LIN {X 0,Y 523.367,Z 631.707,A -85,B 0,C 180,E1 -4773.079,E2 -4773.079} C_VEL
LIN {X 0,Y 523.424,Z 628.783,A -85,B 0,C 180,E1 -4774.235,E2 -4774.235} C_VEL
LIN {X 0,Y 523.464,Z 624.823,A -85,B 0,C 180,E1 -4775.393,E2 -4775.393} C_VEL
LIN {X 0,Y 523.519,Z 619.605,A -85,B 0,C 180,E1 -4776.577,E2 -4776.577} C_VEL
LIN {X 0,Y 523.664,Z 613.306,A -85,B 0,C 180,E1 -4777.713,E2 -4777.713} C_VEL
LIN {X 0,Y 523.85,Z 605.295,A -85,B 0,C 180,E1 -4778.875,E2 -4778.875} C_VEL
LIN {X 0,Y 524.066,Z 597.13,A -85,B 0,C 180,E1 -4779.845,E2 -4779.845} C_VEL
LIN {X 0,Y 524.349,Z 587.171,A -85,B 0,C 180,E1 -4780.815,E2 -4780.815} C_VEL
LIN {X 0,Y 524.625,Z 575.842,A -85,B 0,C 180,E1 -4781.695,E2 -4781.695} C_VEL
LIN {X 0,Y 524.913,Z 564.896,A -85,B 0,C 180,E1 -4782.37,E2 -4782.37} C_VEL
LIN {X 0,Y 525.171,Z 552.673,A -85,B 0,C 180,E1 -4782.953,E2 -4782.953} C_VEL
LIN {X 0,Y 525.375,Z 539.835,A -85,B 0,C 180,E1 -4783.391,E2 -4783.391} C_VEL
LIN {X 0,Y 525.592,Z 526.212,A -85,B 0,C 180,E1 -4783.681,E2 -4783.681} C_VEL
LIN {X 0,Y 525.826,Z 432.447,A -85,B 0,C 180,E1 -4784.974,E2 -4784.974} C_VEL
LIN {X 0,Y 524.297,Z 423.023,A -85,B 0,C 180,E1 -4785.174,E2 -4785.174} C_VEL
LIN {X 0,Y 524.677,Z 405.609,A -85,B 0,C 180,E1 -4788.003,E2 -4788.003} C_VEL
LIN {X 0,Y 525.177,Z 385.391,A -85,B 0,C 180,E1 -4791.387,E2 -4791.387} C_VEL
LIN {X 0,Y 525.133,Z 380.293,A -85,B 0,C 180,E1 -4792.258,E2 -4792.258} C_VEL
LIN {X 0,Y 523.971,Z 373.816,A -85,B 0,C 180,E1 -4793.465,E2 -4793.465} C_VEL
LIN {X 0,Y 523.976,Z 373.714,A -85,B 0,C 180,E1 -4796.271,E2 -4796.271} C_VEL
LIN {X 0,Y 523.956,Z 373.722,A -85,B 0,C 180,E1 -4799.323,E2 -4799.323} C_VEL
LIN {X 0,Y 523.941,Z 373.716,A -85,B 0,C 180,E1 -4802.449,E2 -4802.449} C_VEL
LIN {X 0,Y 523.936,Z 373.723,A -85,B 0,C 180,E1 -4805.225,E2 -4805.225} C_VEL
LIN {X 0,Y 523.919,Z 373.719,A -85,B 0,C 180,E1 -4808.101,E2 -4808.101} C_VEL
LIN {X 0,Y 523.961,Z 373.722,A -85,B 0,C 180,E1 -4811.31,E2 -4811.31} C_VEL
LIN {X 0,Y 523.954,Z 373.717,A -85,B 0,C 180,E1 -4814.691,E2 -4814.691} C_VEL
LIN {X 0,Y 523.964,Z 373.714,A -85,B 0,C 180,E1 -4817.882,E2 -4817.882} C_VEL
LIN {X 0,Y 523.957,Z 373.72,A -85,B 0,C 180,E1 -4820.918,E2 -4820.918} C_VEL
LIN {X 0,Y 523.925,Z 373.719,A -85,B 0,C 180,E1 -4823.827,E2 -4823.827} C_VEL
LIN {X 0,Y 523.939,Z 373.721,A -85,B 0,C 180,E1 -4826.635,E2 -4826.635} C_VEL
LIN {X 0,Y 523.952,Z 373.719,A -85,B 0,C 180,E1 -4829.355,E2 -4829.355} C_VEL
LIN {X 0,Y 523.975,Z 373.714,A -85,B 0,C 180,E1 -4832.28,E2 -4832.28} C_VEL
LIN {X 0,Y 523.95,Z 373.72,A -85,B 0,C 180,E1 -4834.581,E2 -4834.581} C_VEL
LIN {X 0,Y 523.911,Z 373.726,A -85,B 0,C 180,E1 -4837.106,E2 -4837.106} C_VEL
LIN {X 0,Y 523.973,Z 373.713,A -85,B 0,C 180,E1 -4839.865,E2 -4839.865} C_VEL
LIN {X 0,Y 523.965,Z 373.721,A -85,B 0,C 180,E1 -4842.837,E2 -4842.837} C_VEL
LIN {X 0,Y 523.97,Z 373.715,A -85,B 0,C 180,E1 -4845.235,E2 -4845.235} C_VEL
LIN {X 0,Y 524.006,Z 373.714,A -85,B 0,C 180,E1 -4848.394,E2 -4848.394} C_VEL
LIN {X 0,Y 523.999,Z 373.71,A -85,B 0,C 180,E1 -4851.516,E2 -4851.516} C_VEL
LIN {X 0,Y 524.077,Z 373.706,A -85,B 0,C 180,E1 -4854.614,E2 -4854.614} C_VEL
LIN {X 0,Y 524.105,Z 373.698,A -85,B 0,C 180,E1 -4857.694,E2 -4857.694} C_VEL
LIN {X 0,Y 524.118,Z 373.699,A -85,B 0,C 180,E1 -4860.768,E2 -4860.768} C_VEL
LIN {X 0,Y 524.069,Z 373.702,A -85,B 0,C 180,E1 -4863.075,E2 -4863.075} C_VEL
LIN {X 0,Y 524.04,Z 373.71,A -85,B 0,C 180,E1 -4866.159,E2 -4866.159} C_VEL
LIN {X 0,Y 523.994,Z 373.711,A -85,B 0,C 180,E1 -4869.262,E2 -4869.262} C_VEL
LIN {X 0,Y 523.996,Z 373.714,A -85,B 0,C 180,E1 -4871.74,E2 -4871.74} C_VEL
LIN {X 0,Y 523.986,Z 373.712,A -85,B 0,C 180,E1 -4875.052,E2 -4875.052} C_VEL
LIN {X 0,Y 523.958,Z 373.721,A -85,B 0,C 180,E1 -4877.969,E2 -4877.969} C_VEL
LIN {X 0,Y 523.967,Z 373.718,A -85,B 0,C 180,E1 -4880.41,E2 -4880.41} C_VEL
LIN {X 0,Y 523.911,Z 373.721,A -85,B 0,C 180,E1 -4882.894,E2 -4882.894} C_VEL
LIN {X 0,Y 523.95,Z 373.719,A -85,B 0,C 180,E1 -4885.419,E2 -4885.419} C_VEL
LIN {X 0,Y 523.966,Z 373.719,A -85,B 0,C 180,E1 -4887.999,E2 -4887.999} C_VEL
LIN {X 0,Y 523.948,Z 373.717,A -85,B 0,C 180,E1 -4890.857,E2 -4890.857} C_VEL
LIN {X 0,Y 523.958,Z 373.721,A -85,B 0,C 180,E1 -4893.736,E2 -4893.736} C_VEL
LIN {X 0,Y 523.919,Z 373.721,A -85,B 0,C 180,E1 -4896.405,E2 -4896.405} C_VEL
LIN {X 0,Y 523.92,Z 373.721,A -85,B 0,C 180,E1 -4899.085,E2 -4899.085} C_VEL
LIN {X 0,Y 523.954,Z 373.718,A -85,B 0,C 180,E1 -4902.119,E2 -4902.119} C_VEL
LIN {X 0,Y 523.953,Z 373.721,A -85,B 0,C 180,E1 -4905.309,E2 -4905.309} C_VEL
LIN {X 0,Y 523.917,Z 373.721,A -85,B 0,C 180,E1 -4906.922,E2 -4906.922} C_VEL
LIN {X 0,Y 523.255,Z 373.808,A -85,B 0,C 180,E1 -4907.564,E2 -4907.564} C_VEL
LIN {X 0,Y 520.427,Z 374.158,A -85,B 0,C 180,E1 -4908.606,E2 -4908.606} C_VEL
LIN {X 0,Y 518.029,Z 374.46,A -85,B 0,C 180,E1 -4909.445,E2 -4909.445} C_VEL
LIN {X 0,Y 516.99,Z 374.584,A -85,B 0,C 180,E1 -4910.093,E2 -4910.093} C_VEL
LIN {X 0,Y 516.9,Z 374.594,A -85,B 0,C 180,E1 -4910.312,E2 -4910.312} C_VEL
LIN {X 0,Y 516.884,Z 374.603,A -85,B 0,C 180,E1 -4913.342,E2 -4913.342} C_VEL
LIN {X 0,Y 516.912,Z 374.593,A -85,B 0,C 180,E1 -4916.122,E2 -4916.122} C_VEL
LIN {X 0,Y 516.891,Z 374.599,A -85,B 0,C 180,E1 -4918.936,E2 -4918.936} C_VEL
LIN {X 0,Y 516.919,Z 374.595,A -85,B 0,C 180,E1 -4921.585,E2 -4921.585} C_VEL
LIN {X 0,Y 516.932,Z 374.59,A -85,B 0,C 180,E1 -4924.211,E2 -4924.211} C_VEL
LIN {X 0,Y 516.866,Z 374.601,A -85,B 0,C 180,E1 -4926.777,E2 -4926.777} C_VEL
LIN {X 0,Y 516.94,Z 374.59,A -85,B 0,C 180,E1 -4929.732,E2 -4929.732} C_VEL
LIN {X 0,Y 516.923,Z 374.593,A -85,B 0,C 180,E1 -4932.596,E2 -4932.596} C_VEL
LIN {X 0,Y 516.944,Z 374.596,A -85,B 0,C 180,E1 -4935.03,E2 -4935.03} C_VEL
LIN {X 0,Y 516.968,Z 374.588,A -85,B 0,C 180,E1 -4938.234,E2 -4938.234} C_VEL
LIN {X 0,Y 517.009,Z 374.749,A -85,B 0,C 180,E1 -4941.203,E2 -4941.203} C_VEL
LIN {X 0,Y 517.924,Z 380.978,A -85,B 0,C 180,E1 -4942.447,E2 -4942.447} C_VEL
LIN {X 0,Y 517.682,Z 391.15,A -85,B 0,C 180,E1 -4944.351,E2 -4944.351} C_VEL
LIN {X 0,Y 517.287,Z 408.071,A -85,B 0,C 180,E1 -4947.469,E2 -4947.469} C_VEL
LIN {X 0,Y 517.331,Z 409.756,A -85,B 0,C 180,E1 -4947.688,E2 -4947.688} C_VEL
LIN {X 0,Y 519.148,Z 421.04,A -85,B 0,C 180,E1 -4947.915,E2 -4947.915} C_VEL
LIN {X 0,Y 518.607,Z 517.117,A -85,B 0,C 180,E1 -4949.272,E2 -4949.272} C_VEL
LIN {X 0,Y 518.401,Z 530.709,A -85,B 0,C 180,E1 -4949.636,E2 -4949.636} C_VEL
LIN {X 0,Y 518.149,Z 543.463,A -85,B 0,C 180,E1 -4950.146,E2 -4950.146} C_VEL
LIN {X 0,Y 517.833,Z 555.117,A -85,B 0,C 180,E1 -4950.777,E2 -4950.777} C_VEL
LIN {X 0,Y 517.475,Z 566.364,A -85,B 0,C 180,E1 -4951.556,E2 -4951.556} C_VEL
LIN {X 0,Y 517.179,Z 576.521,A -85,B 0,C 180,E1 -4952.434,E2 -4952.434} C_VEL
LIN {X 0,Y 516.891,Z 586.48,A -85,B 0,C 180,E1 -4953.508,E2 -4953.508} C_VEL
LIN {X 0,Y 516.678,Z 595.257,A -85,B 0,C 180,E1 -4954.681,E2 -4954.681} C_VEL
LIN {X 0,Y 516.538,Z 602.327,A -85,B 0,C 180,E1 -4955.857,E2 -4955.857} C_VEL
LIN {X 0,Y 516.391,Z 607.986,A -85,B 0,C 180,E1 -4957.035,E2 -4957.035} C_VEL
LIN {X 0,Y 516.351,Z 612.449,A -85,B 0,C 180,E1 -4958.216,E2 -4958.216} C_VEL
LIN {X 0,Y 516.224,Z 615.851,A -85,B 0,C 180,E1 -4959.402,E2 -4959.402} C_VEL
LIN {X 0,Y 516.247,Z 617.536,A -85,B 0,C 180,E1 -4960.193,E2 -4960.193} C_VEL
LIN {X 0,Y 516.261,Z 619.345,A -85,B 0,C 180,E1 -4961.433,E2 -4961.433} C_VEL
LIN {X 0,Y 516.177,Z 620.126,A -85,B 0,C 180,E1 -4962.582,E2 -4962.582} C_VEL
LIN {X 0,Y 516.167,Z 620.151,A -85,B 0,C 180,E1 -4963.383,E2 -4963.383} C_VEL
LIN {X 0,Y 516.203,Z 619.159,A -85,B 0,C 180,E1 -4964.839,E2 -4964.839} C_VEL
LIN {X 0,Y 516.164,Z 617.713,A -85,B 0,C 180,E1 -4965.802,E2 -4965.802} C_VEL
LIN {X 0,Y 516.263,Z 614.996,A -85,B 0,C 180,E1 -4967.018,E2 -4967.018} C_VEL
LIN {X 0,Y 516.346,Z 611.168,A -85,B 0,C 180,E1 -4968.243,E2 -4968.243} C_VEL
LIN {X 0,Y 516.438,Z 606.1,A -85,B 0,C 180,E1 -4969.475,E2 -4969.475} C_VEL
LIN {X 0,Y 516.563,Z 599.617,A -85,B 0,C 180,E1 -4970.715,E2 -4970.715} C_VEL
LIN {X 0,Y 516.771,Z 592.904,A -85,B 0,C 180,E1 -4971.752,E2 -4971.752} C_VEL
LIN {X 0,Y 517.029,Z 584.057,A -85,B 0,C 180,E1 -4972.866,E2 -4972.866} C_VEL
LIN {X 0,Y 517.298,Z 573.392,A -85,B 0,C 180,E1 -4973.946,E2 -4973.946} C_VEL
LIN {X 0,Y 517.614,Z 563.26,A -85,B 0,C 180,E1 -4974.77,E2 -4974.77} C_VEL
LIN {X 0,Y 517.954,Z 551.645,A -85,B 0,C 180,E1 -4975.518,E2 -4975.518} C_VEL
LIN {X 0,Y 518.219,Z 540.041,A -85,B 0,C 180,E1 -4976.097,E2 -4976.097} C_VEL
LIN {X 0,Y 518.493,Z 527.118,A -85,B 0,C 180,E1 -4976.57,E2 -4976.57} C_VEL
LIN {X 0,Y 518.663,Z 514.974,A -85,B 0,C 180,E1 -4976.859,E2 -4976.859} C_VEL
LIN {X 0,Y 519.104,Z 420.064,A -85,B 0,C 180,E1 -4978.191,E2 -4978.191} C_VEL
LIN {X 0,Y 517.285,Z 409.483,A -85,B 0,C 180,E1 -4978.42,E2 -4978.42} C_VEL
LIN {X 0,Y 517.352,Z 404.526,A -85,B 0,C 180,E1 -4979.277,E2 -4979.277} C_VEL
LIN {X 0,Y 517.808,Z 387.557,A -85,B 0,C 180,E1 -4982.415,E2 -4982.415} C_VEL
LIN {X 0,Y 517.913,Z 380.164,A -85,B 0,C 180,E1 -4983.804,E2 -4983.804} C_VEL
LIN {X 0,Y 516.928,Z 374.673,A -85,B 0,C 180,E1 -4984.937,E2 -4984.937} C_VEL
LIN {X 0,Y 516.882,Z 374.598,A -85,B 0,C 180,E1 -4987.943,E2 -4987.943} C_VEL
LIN {X 0,Y 516.9,Z 374.599,A -85,B 0,C 180,E1 -4990.739,E2 -4990.739} C_VEL
LIN {X 0,Y 516.878,Z 374.598,A -85,B 0,C 180,E1 -4993.902,E2 -4993.902} C_VEL
LIN {X 0,Y 516.878,Z 374.596,A -85,B 0,C 180,E1 -4996.106,E2 -4996.106} C_VEL
LIN {X 0,Y 516.903,Z 374.6,A -85,B 0,C 180,E1 -4999.26,E2 -4999.26} C_VEL
LIN {X 0,Y 516.879,Z 374.595,A -85,B 0,C 180,E1 -5002.055,E2 -5002.055} C_VEL
LIN {X 0,Y 516.89,Z 374.597,A -85,B 0,C 180,E1 -5005.176,E2 -5005.176} C_VEL
LIN {X 0,Y 516.876,Z 374.596,A -85,B 0,C 180,E1 -5007.975,E2 -5007.975} C_VEL
LIN {X 0,Y 516.928,Z 374.588,A -85,B 0,C 180,E1 -5010.696,E2 -5010.696} C_VEL
LIN {X 0,Y 516.936,Z 374.589,A -85,B 0,C 180,E1 -5013.803,E2 -5013.803} C_VEL
LIN {X 0,Y 516.883,Z 374.601,A -85,B 0,C 180,E1 -5016.777,E2 -5016.777} C_VEL
LIN {X 0,Y 516.93,Z 374.59,A -85,B 0,C 180,E1 -5019.731,E2 -5019.731} C_VEL
LIN {X 0,Y 516.922,Z 374.592,A -85,B 0,C 180,E1 -5022.596,E2 -5022.596} C_VEL
LIN {X 0,Y 516.932,Z 374.594,A -85,B 0,C 180,E1 -5025.03,E2 -5025.03} C_VEL
LIN {X 0,Y 516.994,Z 374.582,A -85,B 0,C 180,E1 -5028.234,E2 -5028.234} C_VEL
LIN {X 0,Y 516.964,Z 374.587,A -85,B 0,C 180,E1 -5031.4,E2 -5031.4} C_VEL
LIN {X 0,Y 517.036,Z 374.578,A -85,B 0,C 180,E1 -5034.54,E2 -5034.54} C_VEL
LIN {X 0,Y 517.076,Z 374.57,A -85,B 0,C 180,E1 -5037.663,E2 -5037.663} C_VEL
LIN {X 0,Y 517.088,Z 374.576,A -85,B 0,C 180,E1 -5040.779,E2 -5040.779} C_VEL
LIN {X 0,Y 517.01,Z 374.58,A -85,B 0,C 180,E1 -5043.117,E2 -5043.117} C_VEL
LIN {X 0,Y 517.001,Z 374.582,A -85,B 0,C 180,E1 -5046.243,E2 -5046.243} C_VEL
LIN {X 0,Y 516.95,Z 374.587,A -85,B 0,C 180,E1 -5049.389,E2 -5049.389} C_VEL
LIN {X 0,Y 516.974,Z 374.584,A -85,B 0,C 180,E1 -5051.824,E2 -5051.824} C_VEL
LIN {X 0,Y 516.934,Z 374.592,A -85,B 0,C 180,E1 -5055.147,E2 -5055.147} C_VEL
LIN {X 0,Y 516.917,Z 374.591,A -85,B 0,C 180,E1 -5058.223,E2 -5058.223} C_VEL
LIN {X 0,Y 516.907,Z 374.601,A -85,B 0,C 180,E1 -5060.702,E2 -5060.702} C_VEL
LIN {X 0,Y 516.884,Z 374.596,A -85,B 0,C 180,E1 -5063.223,E2 -5063.223} C_VEL
LIN {X 0,Y 516.937,Z 374.59,A -85,B 0,C 180,E1 -5066.197,E2 -5066.197} C_VEL
LIN {X 0,Y 516.915,Z 374.592,A -85,B 0,C 180,E1 -5069.305,E2 -5069.305} C_VEL
LIN {X 0,Y 516.895,Z 374.602,A -85,B 0,C 180,E1 -5072.545,E2 -5072.545} C_VEL
LIN {X 0,Y 516.878,Z 374.597,A -85,B 0,C 180,E1 -5075.333,E2 -5075.333} C_VEL
LIN {X 0,Y 516.876,Z 374.596,A -85,B 0,C 180,E1 -5077.944,E2 -5077.944} C_VEL
LIN {X 0,Y 516.9,Z 374.593,A -85,B 0,C 180,E1 -5080.74,E2 -5080.74} C_VEL
LIN {X 0,Y 516.878,Z 374.597,A -85,B 0,C 180,E1 -5083.904,E2 -5083.904} C_VEL
LIN {X 0,Y 516.878,Z 374.597,A -85,B 0,C 180,E1 -5086.108,E2 -5086.108} C_VEL
LIN {X 0,Y 516.914,Z 374.598,A -85,B 0,C 180,E1 -5088.399,E2 -5088.399} C_VEL
LIN {X 0,Y 516.88,Z 374.597,A -85,B 0,C 180,E1 -5091.285,E2 -5091.285} C_VEL
LIN {X 0,Y 516.89,Z 374.597,A -85,B 0,C 180,E1 -5094.222,E2 -5094.222} C_VEL
LIN {X 0,Y 516.898,Z 374.596,A -85,B 0,C 180,E1 -5097.054,E2 -5097.054} C_VEL
LIN {X 0,Y 516.892,Z 374.597,A -85,B 0,C 180,E1 -5099.797,E2 -5099.797} C_VEL
LIN {X 0,Y 516.93,Z 374.598,A -85,B 0,C 180,E1 -5102.468,E2 -5102.468} C_VEL
LIN {X 0,Y 516.913,Z 374.597,A -85,B 0,C 180,E1 -5105.073,E2 -5105.073} C_VEL
LIN {X 0,Y 516.956,Z 374.823,A -85,B 0,C 180,E1 -5106.41,E2 -5106.41} C_VEL
LIN {X 0,Y 518.284,Z 382.852,A -85,B 0,C 180,E1 -5107.896,E2 -5107.896} C_VEL
LIN {X 0,Y 517.825,Z 401.003,A -85,B 0,C 180,E1 -5110.991,E2 -5110.991} C_VEL
LIN {X 0,Y 517.377,Z 417.947,A -85,B 0,C 180,E1 -5113.832,E2 -5113.832} C_VEL
LIN {X 0,Y 517.295,Z 423.024,A -85,B 0,C 180,E1 -5114.623,E2 -5114.623} C_VEL
LIN {X 0,Y 519.019,Z 433.654,A -85,B 0,C 180,E1 -5114.844,E2 -5114.844} C_VEL
LIN {X 0,Y 518.657,Z 530.448,A -85,B 0,C 180,E1 -5116.208,E2 -5116.208} C_VEL
LIN {X 0,Y 518.394,Z 543.764,A -85,B 0,C 180,E1 -5116.551,E2 -5116.551} C_VEL
LIN {X 0,Y 518.097,Z 557.071,A -85,B 0,C 180,E1 -5117.067,E2 -5117.067} C_VEL
LIN {X 0,Y 517.842,Z 569.422,A -85,B 0,C 180,E1 -5117.733,E2 -5117.733} C_VEL
LIN {X 0,Y 517.52,Z 581.126,A -85,B 0,C 180,E1 -5118.545,E2 -5118.545} C_VEL
LIN {X 0,Y 517.191,Z 591.315,A -85,B 0,C 180,E1 -5119.43,E2 -5119.43} C_VEL
LIN {X 0,Y 516.954,Z 600.48,A -85,B 0,C 180,E1 -5120.414,E2 -5120.414} C_VEL
LIN {X 0,Y 516.71,Z 609.408,A -85,B 0,C 180,E1 -5121.593,E2 -5121.593} C_VEL
LIN {X 0,Y 516.51,Z 616.591,A -85,B 0,C 180,E1 -5122.77,E2 -5122.77} C_VEL
LIN {X 0,Y 516.435,Z 623.131,A -85,B 0,C 180,E1 -5124.142,E2 -5124.142} C_VEL
LIN {X 0,Y 516.271,Z 627.456,A -85,B 0,C 180,E1 -5125.315,E2 -5125.315} C_VEL
LIN {X 0,Y 516.352,Z 629.746,A -85,B 0,C 180,E1 -5126.098,E2 -5126.098} C_VEL
LIN {X 0,Y 516.282,Z 631.601,A -85,B 0,C 180,E1 -5126.879,E2 -5126.879} C_VEL
LIN {X 0,Y 516.261,Z 632.992,A -85,B 0,C 180,E1 -5127.66,E2 -5127.66} C_VEL
LIN {X 0,Y 516.16,Z 634.59,A -85,B 0,C 180,E1 -5129.22,E2 -5129.22} C_VEL
LIN {X 0,Y 516.154,Z 634.806,A -85,B 0,C 180,E1 -5130,E2 -5130} C_VEL
LIN {X 0,Y 516.192,Z 633.987,A -85,B 0,C 180,E1 -5131.561,E2 -5131.561} C_VEL
LIN {X 0,Y 516.261,Z 632.996,A -85,B 0,C 180,E1 -5132.341,E2 -5132.341} C_VEL
LIN {X 0,Y 516.282,Z 631.606,A -85,B 0,C 180,E1 -5133.121,E2 -5133.121} C_VEL
LIN {X 0,Y 516.314,Z 628.681,A -85,B 0,C 180,E1 -5134.294,E2 -5134.294} C_VEL
LIN {X 0,Y 516.402,Z 624.721,A -85,B 0,C 180,E1 -5135.467,E2 -5135.467} C_VEL
LIN {X 0,Y 516.482,Z 618.813,A -85,B 0,C 180,E1 -5136.802,E2 -5136.802} C_VEL
LIN {X 0,Y 516.635,Z 611.968,A -85,B 0,C 180,E1 -5138.015,E2 -5138.015} C_VEL
LIN {X 0,Y 516.852,Z 603.702,A -85,B 0,C 180,E1 -5139.194,E2 -5139.194} C_VEL
LIN {X 0,Y 517.078,Z 595.226,A -85,B 0,C 180,E1 -5140.177,E2 -5140.177} C_VEL
LIN {X 0,Y 517.405,Z 584.75,A -85,B 0,C 180,E1 -5141.161,E2 -5141.161} C_VEL
LIN {X 0,Y 517.752,Z 573.003,A -85,B 0,C 180,E1 -5142.043,E2 -5142.043} C_VEL
LIN {X 0,Y 518.033,Z 561.086,A -85,B 0,C 180,E1 -5142.736,E2 -5142.736} C_VEL
LIN {X 0,Y 518.338,Z 548.735,A -85,B 0,C 180,E1 -5143.276,E2 -5143.276} C_VEL
LIN {X 0,Y 518.568,Z 536.047,A -85,B 0,C 180,E1 -5143.67,E2 -5143.67} C_VEL
LIN {X 0,Y 518.719,Z 520.963,A -85,B 0,C 180,E1 -5143.94,E2 -5143.94} C_VEL
LIN {X 0,Y 518.993,Z 433.377,A -85,B 0,C 180,E1 -5145.161,E2 -5145.161} C_VEL
LIN {X 0,Y 517.303,Z 422.955,A -85,B 0,C 180,E1 -5145.382,E2 -5145.382} C_VEL
LIN {X 0,Y 517.702,Z 406.165,A -85,B 0,C 180,E1 -5148.143,E2 -5148.143} C_VEL
LIN {X 0,Y 518.217,Z 386.518,A -85,B 0,C 180,E1 -5151.479,E2 -5151.479} C_VEL
LIN {X 0,Y 518.189,Z 381.679,A -85,B 0,C 180,E1 -5152.318,E2 -5152.318} C_VEL
LIN {X 0,Y 516.957,Z 374.806,A -85,B 0,C 180,E1 -5153.59,E2 -5153.59} C_VEL
LIN {X 0,Y 516.928,Z 374.591,A -85,B 0,C 180,E1 -5156.657,E2 -5156.657} C_VEL
LIN {X 0,Y 516.912,Z 374.6,A -85,B 0,C 180,E1 -5159.523,E2 -5159.523} C_VEL
LIN {X 0,Y 516.901,Z 374.593,A -85,B 0,C 180,E1 -5162.544,E2 -5162.544} C_VEL
LIN {X 0,Y 516.884,Z 374.603,A -85,B 0,C 180,E1 -5165.332,E2 -5165.332} C_VEL
LIN {X 0,Y 516.884,Z 374.597,A -85,B 0,C 180,E1 -5167.943,E2 -5167.943} C_VEL
LIN {X 0,Y 516.885,Z 374.597,A -85,B 0,C 180,E1 -5170.741,E2 -5170.741} C_VEL
LIN {X 0,Y 516.903,Z 374.596,A -85,B 0,C 180,E1 -5172.829,E2 -5172.829} C_VEL
LIN {X 0,Y 516.921,Z 374.596,A -85,B 0,C 180,E1 -5175.009,E2 -5175.009} C_VEL
LIN {X 0,Y 516.927,Z 374.591,A -85,B 0,C 180,E1 -5178.396,E2 -5178.396} C_VEL
LIN {X 0,Y 516.903,Z 374.6,A -85,B 0,C 180,E1 -5181.286,E2 -5181.286} C_VEL
LIN {X 0,Y 516.887,Z 374.596,A -85,B 0,C 180,E1 -5184.221,E2 -5184.221} C_VEL
LIN {X 0,Y 516.894,Z 374.602,A -85,B 0,C 180,E1 -5187.053,E2 -5187.053} C_VEL
LIN {X 0,Y 516.888,Z 374.596,A -85,B 0,C 180,E1 -5189.796,E2 -5189.796} C_VEL
LIN {X 0,Y 516.926,Z 374.594,A -85,B 0,C 180,E1 -5192.467,E2 -5192.467} C_VEL
LIN {X 0,Y 516.907,Z 374.599,A -85,B 0,C 180,E1 -5195.072,E2 -5195.072} C_VEL
LIN {X 0,Y 516.881,Z 374.601,A -85,B 0,C 180,E1 -5198.462,E2 -5198.462} C_VEL
LIN {X 0,Y 516.9,Z 374.6,A -85,B 0,C 180,E1 -5200.955,E2 -5200.955} C_VEL
LIN {X 0,Y 516.911,Z 374.594,A -85,B 0,C 180,E1 -5203.41,E2 -5203.41} C_VEL
LIN {X 0,Y 516.889,Z 374.596,A -85,B 0,C 180,E1 -5205.833,E2 -5205.833} C_VEL
LIN {X 0,Y 516.959,Z 374.591,A -85,B 0,C 180,E1 -5208.233,E2 -5208.233} C_VEL
LIN {X 0,Y 516.963,Z 374.587,A -85,B 0,C 180,E1 -5211.399,E2 -5211.399} C_VEL
LIN {X 0,Y 517.003,Z 374.583,A -85,B 0,C 180,E1 -5213.757,E2 -5213.757} C_VEL
LIN {X 0,Y 517.077,Z 374.573,A -85,B 0,C 180,E1 -5217.663,E2 -5217.663} C_VEL
LIN {X 0,Y 517.088,Z 374.575,A -85,B 0,C 180,E1 -5220.779,E2 -5220.779} C_VEL
LIN {X 0,Y 517.01,Z 374.582,A -85,B 0,C 180,E1 -5223.117,E2 -5223.117} C_VEL
LIN {X 0,Y 517.004,Z 374.586,A -85,B 0,C 180,E1 -5226.243,E2 -5226.243} C_VEL
LIN {X 0,Y 516.948,Z 374.589,A -85,B 0,C 180,E1 -5229.389,E2 -5229.389} C_VEL
LIN {X 0,Y 516.945,Z 374.593,A -85,B 0,C 180,E1 -5231.807,E2 -5231.807} C_VEL
LIN {X 0,Y 516.937,Z 374.59,A -85,B 0,C 180,E1 -5235.147,E2 -5235.147} C_VEL
LIN {X 0,Y 516.92,Z 374.597,A -85,B 0,C 180,E1 -5238.222,E2 -5238.222} C_VEL
LIN {X 0,Y 516.907,Z 374.595,A -85,B 0,C 180,E1 -5240.702,E2 -5240.702} C_VEL
LIN {X 0,Y 516.906,Z 374.598,A -85,B 0,C 180,E1 -5244.072,E2 -5244.072} C_VEL
LIN {X 0,Y 516.924,Z 374.592,A -85,B 0,C 180,E1 -5246.658,E2 -5246.658} C_VEL
LIN {X 0,Y 516.92,Z 374.597,A -85,B 0,C 180,E1 -5249.527,E2 -5249.527} C_VEL
LIN {X 0,Y 516.897,Z 374.596,A -85,B 0,C 180,E1 -5252.545,E2 -5252.545} C_VEL
LIN {X 0,Y 516.879,Z 374.6,A -85,B 0,C 180,E1 -5255.333,E2 -5255.333} C_VEL
LIN {X 0,Y 516.878,Z 374.601,A -85,B 0,C 180,E1 -5257.944,E2 -5257.944} C_VEL
LIN {X 0,Y 516.882,Z 374.597,A -85,B 0,C 180,E1 -5260.742,E2 -5260.742} C_VEL
LIN {X 0,Y 516.902,Z 374.595,A -85,B 0,C 180,E1 -5262.83,E2 -5262.83} C_VEL
LIN {X 0,Y 516.92,Z 374.594,A -85,B 0,C 180,E1 -5265.011,E2 -5265.011} C_VEL
LIN {X 0,Y 516.921,Z 374.592,A -85,B 0,C 180,E1 -5268.398,E2 -5268.398} C_VEL
LIN {X 0,Y 516.9,Z 374.594,A -85,B 0,C 180,E1 -5270.312,E2 -5270.312} C_VEL
LIN {X 0,Y 516.22,Z 374.682,A -85,B 0,C 180,E1 -5270.962,E2 -5270.962} C_VEL
LIN {X 0,Y 513.366,Z 375.04,A -85,B 0,C 180,E1 -5272.018,E2 -5272.018} C_VEL
LIN {X 0,Y 510.957,Z 375.342,A -85,B 0,C 180,E1 -5272.868,E2 -5272.868} C_VEL
LIN {X 0,Y 509.918,Z 375.469,A -85,B 0,C 180,E1 -5273.524,E2 -5273.524} C_VEL
LIN {X 0,Y 509.83,Z 375.478,A -85,B 0,C 180,E1 -5273.746,E2 -5273.746} C_VEL
LIN {X 0,Y 509.862,Z 375.471,A -85,B 0,C 180,E1 -5276.54,E2 -5276.54} C_VEL
LIN {X 0,Y 509.845,Z 375.479,A -85,B 0,C 180,E1 -5279.335,E2 -5279.335} C_VEL
LIN {X 0,Y 509.892,Z 375.467,A -85,B 0,C 180,E1 -5282.055,E2 -5282.055} C_VEL
LIN {X 0,Y 509.877,Z 375.471,A -85,B 0,C 180,E1 -5284.704,E2 -5284.704} C_VEL
LIN {X 0,Y 509.828,Z 375.478,A -85,B 0,C 180,E1 -5287.458,E2 -5287.458} C_VEL
LIN {X 0,Y 509.918,Z 375.464,A -85,B 0,C 180,E1 -5289.845,E2 -5289.845} C_VEL
LIN {X 0,Y 509.883,Z 375.474,A -85,B 0,C 180,E1 -5293.175,E2 -5293.175} C_VEL
LIN {X 0,Y 509.866,Z 375.472,A -85,B 0,C 180,E1 -5295.634,E2 -5295.634} C_VEL
LIN {X 0,Y 509.916,Z 375.471,A -85,B 0,C 180,E1 -5298.875,E2 -5298.875} C_VEL
LIN {X 0,Y 509.966,Z 375.582,A -85,B 0,C 180,E1 -5301.031,E2 -5301.031} C_VEL
LIN {X 0,Y 510.97,Z 382.117,A -85,B 0,C 180,E1 -5302.358,E2 -5302.358} C_VEL
LIN {X 0,Y 510.706,Z 392.236,A -85,B 0,C 180,E1 -5304.274,E2 -5304.274} C_VEL
LIN {X 0,Y 510.3,Z 408.654,A -85,B 0,C 180,E1 -5307.336,E2 -5307.336} C_VEL
LIN {X 0,Y 510.308,Z 409.616,A -85,B 0,C 180,E1 -5307.459,E2 -5307.459} C_VEL
LIN {X 0,Y 512.316,Z 421.607,A -85,B 0,C 180,E1 -5307.715,E2 -5307.715} C_VEL
LIN {X 0,Y 511.741,Z 516.369,A -85,B 0,C 180,E1 -5309.065,E2 -5309.065} C_VEL
LIN {X 0,Y 511.553,Z 529.479,A -85,B 0,C 180,E1 -5309.409,E2 -5309.409} C_VEL
LIN {X 0,Y 511.273,Z 542.093,A -85,B 0,C 180,E1 -5309.901,E2 -5309.901} C_VEL
LIN {X 0,Y 510.953,Z 553.351,A -85,B 0,C 180,E1 -5310.492,E2 -5310.492} C_VEL
LIN {X 0,Y 510.563,Z 564.952,A -85,B 0,C 180,E1 -5311.282,E2 -5311.282} C_VEL
LIN {X 0,Y 510.258,Z 575.365,A -85,B 0,C 180,E1 -5312.17,E2 -5312.17} C_VEL
LIN {X 0,Y 509.929,Z 584.799,A -85,B 0,C 180,E1 -5313.16,E2 -5313.16} C_VEL
LIN {X 0,Y 509.695,Z 593.886,A -85,B 0,C 180,E1 -5314.349,E2 -5314.349} C_VEL
LIN {X 0,Y 509.44,Z 601.24,A -85,B 0,C 180,E1 -5315.541,E2 -5315.541} C_VEL
LIN {X 0,Y 509.374,Z 607.138,A -85,B 0,C 180,E1 -5316.734,E2 -5316.734} C_VEL
LIN {X 0,Y 509.277,Z 611.821,A -85,B 0,C 180,E1 -5317.932,E2 -5317.932} C_VEL
LIN {X 0,Y 509.175,Z 615.405,A -85,B 0,C 180,E1 -5319.133,E2 -5319.133} C_VEL
LIN {X 0,Y 509.145,Z 617.971,A -85,B 0,C 180,E1 -5320.337,E2 -5320.337} C_VEL
LIN {X 0,Y 509.168,Z 619.51,A -85,B 0,C 180,E1 -5321.476,E2 -5321.476} C_VEL
LIN {X 0,Y 509.081,Z 620.263,A -85,B 0,C 180,E1 -5322.761,E2 -5322.761} C_VEL
LIN {X 0,Y 509.077,Z 620.214,A -85,B 0,C 180,E1 -5323.573,E2 -5323.573} C_VEL
LIN {X 0,Y 509.118,Z 619.205,A -85,B 0,C 180,E1 -5324.917,E2 -5324.917} C_VEL
LIN {X 0,Y 509.074,Z 617.471,A -85,B 0,C 180,E1 -5326.028,E2 -5326.028} C_VEL
LIN {X 0,Y 509.194,Z 614.592,A -85,B 0,C 180,E1 -5327.262,E2 -5327.262} C_VEL
LIN {X 0,Y 509.275,Z 610.589,A -85,B 0,C 180,E1 -5328.505,E2 -5328.505} C_VEL
LIN {X 0,Y 509.4,Z 605.332,A -85,B 0,C 180,E1 -5329.755,E2 -5329.755} C_VEL
LIN {X 0,Y 509.528,Z 598.573,A -85,B 0,C 180,E1 -5331.015,E2 -5331.015} C_VEL
LIN {X 0,Y 509.802,Z 590.283,A -85,B 0,C 180,E1 -5332.244,E2 -5332.244} C_VEL
LIN {X 0,Y 510.099,Z 581.192,A -85,B 0,C 180,E1 -5333.334,E2 -5333.334} C_VEL
LIN {X 0,Y 510.401,Z 571.314,A -85,B 0,C 180,E1 -5334.29,E2 -5334.29} C_VEL
LIN {X 0,Y 510.761,Z 560.038,A -85,B 0,C 180,E1 -5335.165,E2 -5335.165} C_VEL
LIN {X 0,Y 511.052,Z 548.243,A -85,B 0,C 180,E1 -5335.888,E2 -5335.888} C_VEL
LIN {X 0,Y 511.429,Z 535.832,A -85,B 0,C 180,E1 -5336.454,E2 -5336.454} C_VEL
LIN {X 0,Y 511.652,Z 522.895,A -85,B 0,C 180,E1 -5336.875,E2 -5336.875} C_VEL
LIN {X 0,Y 511.816,Z 509.542,A -85,B 0,C 180,E1 -5337.138,E2 -5337.138} C_VEL
LIN {X 0,Y 512.27,Z 420.85,A -85,B 0,C 180,E1 -5338.388,E2 -5338.388} C_VEL
LIN {X 0,Y 510.297,Z 409.598,A -85,B 0,C 180,E1 -5338.635,E2 -5338.635} C_VEL
LIN {X 0,Y 510.381,Z 404.706,A -85,B 0,C 180,E1 -5339.49,E2 -5339.49} C_VEL
LIN {X 0,Y 510.891,Z 387.577,A -85,B 0,C 180,E1 -5342.702,E2 -5342.702} C_VEL
LIN {X 0,Y 510.968,Z 381.564,A -85,B 0,C 180,E1 -5343.851,E2 -5343.851} C_VEL
LIN {X 0,Y 509.87,Z 375.535,A -85,B 0,C 180,E1 -5345.117,E2 -5345.117} C_VEL
LIN {X 0,Y 509.857,Z 375.473,A -85,B 0,C 180,E1 -5348.336,E2 -5348.336} C_VEL
LIN {X 0,Y 509.862,Z 375.477,A -85,B 0,C 180,E1 -5351.424,E2 -5351.424} C_VEL
LIN {X 0,Y 509.851,Z 375.475,A -85,B 0,C 180,E1 -5354.667,E2 -5354.667} C_VEL
LIN {X 0,Y 509.881,Z 375.465,A -85,B 0,C 180,E1 -5358.099,E2 -5358.099} C_VEL
LIN {X 0,Y 509.871,Z 375.472,A -85,B 0,C 180,E1 -5360.65,E2 -5360.65} C_VEL
LIN {X 0,Y 509.83,Z 375.475,A -85,B 0,C 180,E1 -5363.647,E2 -5363.647} C_VEL
LIN {X 0,Y 509.856,Z 375.47,A -85,B 0,C 180,E1 -5366.539,E2 -5366.539} C_VEL
LIN {X 0,Y 509.843,Z 375.471,A -85,B 0,C 180,E1 -5369.334,E2 -5369.334} C_VEL
LIN {X 0,Y 509.888,Z 375.466,A -85,B 0,C 180,E1 -5372.054,E2 -5372.054} C_VEL
LIN {X 0,Y 509.871,Z 375.473,A -85,B 0,C 180,E1 -5374.704,E2 -5374.704} C_VEL
LIN {X 0,Y 509.857,Z 375.471,A -85,B 0,C 180,E1 -5377.447,E2 -5377.447} C_VEL
LIN {X 0,Y 509.908,Z 375.464,A -85,B 0,C 180,E1 -5379.844,E2 -5379.844} C_VEL
LIN {X 0,Y 509.879,Z 375.473,A -85,B 0,C 180,E1 -5383.175,E2 -5383.175} C_VEL
LIN {X 0,Y 509.855,Z 375.469,A -85,B 0,C 180,E1 -5385.634,E2 -5385.634} C_VEL
LIN {X 0,Y 509.916,Z 375.469,A -85,B 0,C 180,E1 -5388.875,E2 -5388.875} C_VEL
LIN {X 0,Y 509.943,Z 375.46,A -85,B 0,C 180,E1 -5392.078,E2 -5392.078} C_VEL
LIN {X 0,Y 509.985,Z 375.455,A -85,B 0,C 180,E1 -5394.464,E2 -5394.464} C_VEL
LIN {X 0,Y 510.048,Z 375.446,A -85,B 0,C 180,E1 -5397.631,E2 -5397.631} C_VEL
LIN {X 0,Y 510.058,Z 375.452,A -85,B 0,C 180,E1 -5400.79,E2 -5400.79} C_VEL
LIN {X 0,Y 509.952,Z 375.459,A -85,B 0,C 180,E1 -5403.16,E2 -5403.16} C_VEL
LIN {X 0,Y 509.969,Z 375.459,A -85,B 0,C 180,E1 -5406.33,E2 -5406.33} C_VEL
LIN {X 0,Y 509.91,Z 375.468,A -85,B 0,C 180,E1 -5408.72,E2 -5408.72} C_VEL
LIN {X 0,Y 509.942,Z 375.46,A -85,B 0,C 180,E1 -5411.931,E2 -5411.931} C_VEL
LIN {X 0,Y 509.884,Z 375.469,A -85,B 0,C 180,E1 -5415.242,E2 -5415.242} C_VEL
LIN {X 0,Y 509.88,Z 375.466,A -85,B 0,C 180,E1 -5418.002,E2 -5418.002} C_VEL
LIN {X 0,Y 509.849,Z 375.475,A -85,B 0,C 180,E1 -5421.002,E2 -5421.002} C_VEL
LIN {X 0,Y 509.842,Z 375.471,A -85,B 0,C 180,E1 -5423.563,E2 -5423.563} C_VEL
LIN {X 0,Y 509.906,Z 375.469,A -85,B 0,C 180,E1 -5426.38,E2 -5426.38} C_VEL
LIN {X 0,Y 509.87,Z 375.474,A -85,B 0,C 180,E1 -5428.845,E2 -5428.845} C_VEL
LIN {X 0,Y 509.818,Z 375.475,A -85,B 0,C 180,E1 -5431.59,E2 -5431.59} C_VEL
LIN {X 0,Y 509.848,Z 375.477,A -85,B 0,C 180,E1 -5434.414,E2 -5434.414} C_VEL
LIN {X 0,Y 509.814,Z 375.475,A -85,B 0,C 180,E1 -5437.341,E2 -5437.341} C_VEL
LIN {X 0,Y 509.856,Z 375.477,A -85,B 0,C 180,E1 -5440.381,E2 -5440.381} C_VEL
LIN {X 0,Y 509.835,Z 375.475,A -85,B 0,C 180,E1 -5443.065,E2 -5443.065} C_VEL
LIN {X 0,Y 509.826,Z 375.473,A -85,B 0,C 180,E1 -5445.793,E2 -5445.793} C_VEL
LIN {X 0,Y 509.855,Z 375.478,A -85,B 0,C 180,E1 -5448.576,E2 -5448.576} C_VEL
LIN {X 0,Y 509.849,Z 375.473,A -85,B 0,C 180,E1 -5451.787,E2 -5451.787} C_VEL
LIN {X 0,Y 509.846,Z 375.479,A -85,B 0,C 180,E1 -5454.624,E2 -5454.624} C_VEL
LIN {X 0,Y 509.866,Z 375.471,A -85,B 0,C 180,E1 -5457.482,E2 -5457.482} C_VEL
LIN {X 0,Y 509.858,Z 375.477,A -85,B 0,C 180,E1 -5460.274,E2 -5460.274} C_VEL
LIN {X 0,Y 509.888,Z 375.471,A -85,B 0,C 180,E1 -5462.945,E2 -5462.945} C_VEL
LIN {X 0,Y 509.885,Z 375.549,A -85,B 0,C 180,E1 -5466.17,E2 -5466.17} C_VEL
LIN {X 0,Y 511.326,Z 384.015,A -85,B 0,C 180,E1 -5467.792,E2 -5467.792} C_VEL
LIN {X 0,Y 510.863,Z 399.701,A -85,B 0,C 180,E1 -5470.513,E2 -5470.513} C_VEL
LIN {X 0,Y 510.419,Z 416.635,A -85,B 0,C 180,E1 -5473.399,E2 -5473.399} C_VEL
LIN {X 0,Y 510.276,Z 422.793,A -85,B 0,C 180,E1 -5474.398,E2 -5474.398} C_VEL
LIN {X 0,Y 512.22,Z 435.135,A -85,B 0,C 180,E1 -5474.661,E2 -5474.661} C_VEL
LIN {X 0,Y 511.774,Z 530.306,A -85,B 0,C 180,E1 -5476.019,E2 -5476.019} C_VEL
LIN {X 0,Y 511.484,Z 543.635,A -85,B 0,C 180,E1 -5476.366,E2 -5476.366} C_VEL
LIN {X 0,Y 511.191,Z 556.95,A -85,B 0,C 180,E1 -5476.889,E2 -5476.889} C_VEL
LIN {X 0,Y 510.879,Z 569.31,A -85,B 0,C 180,E1 -5477.563,E2 -5477.563} C_VEL
LIN {X 0,Y 510.549,Z 581.012,A -85,B 0,C 180,E1 -5478.386,E2 -5478.386} C_VEL
LIN {X 0,Y 510.198,Z 591.204,A -85,B 0,C 180,E1 -5479.283,E2 -5479.283} C_VEL
LIN {X 0,Y 509.918,Z 600.371,A -85,B 0,C 180,E1 -5480.28,E2 -5480.28} C_VEL
LIN {X 0,Y 509.654,Z 609.301,A -85,B 0,C 180,E1 -5481.475,E2 -5481.475} C_VEL
LIN {X 0,Y 509.436,Z 616.485,A -85,B 0,C 180,E1 -5482.669,E2 -5482.669} C_VEL
LIN {X 0,Y 509.322,Z 621.333,A -85,B 0,C 180,E1 -5483.663,E2 -5483.663} C_VEL
LIN {X 0,Y 509.247,Z 626.044,A -85,B 0,C 180,E1 -5484.854,E2 -5484.854} C_VEL
LIN {X 0,Y 509.246,Z 629.644,A -85,B 0,C 180,E1 -5486.043,E2 -5486.043} C_VEL
LIN {X 0,Y 509.2,Z 631.5,A -85,B 0,C 180,E1 -5486.835,E2 -5486.835} C_VEL
LIN {X 0,Y 509.161,Z 632.891,A -85,B 0,C 180,E1 -5487.627,E2 -5487.627} C_VEL
LIN {X 0,Y 509.073,Z 634.49,A -85,B 0,C 180,E1 -5489.209,E2 -5489.209} C_VEL
LIN {X 0,Y 509.065,Z 634.706,A -85,B 0,C 180,E1 -5490,E2 -5490} C_VEL
LIN {X 0,Y 509.112,Z 633.887,A -85,B 0,C 180,E1 -5491.582,E2 -5491.582} C_VEL
LIN {X 0,Y 509.161,Z 632.896,A -85,B 0,C 180,E1 -5492.373,E2 -5492.373} C_VEL
LIN {X 0,Y 509.2,Z 631.506,A -85,B 0,C 180,E1 -5493.165,E2 -5493.165} C_VEL
LIN {X 0,Y 509.207,Z 628.58,A -85,B 0,C 180,E1 -5494.354,E2 -5494.354} C_VEL
LIN {X 0,Y 509.317,Z 624.62,A -85,B 0,C 180,E1 -5495.543,E2 -5495.543} C_VEL
LIN {X 0,Y 509.404,Z 618.979,A -85,B 0,C 180,E1 -5496.844,E2 -5496.844} C_VEL
LIN {X 0,Y 509.565,Z 611.864,A -85,B 0,C 180,E1 -5498.127,E2 -5498.127} C_VEL
LIN {X 0,Y 509.81,Z 603.597,A -85,B 0,C 180,E1 -5499.322,E2 -5499.322} C_VEL
LIN {X 0,Y 510.059,Z 595.119,A -85,B 0,C 180,E1 -5500.319,E2 -5500.319} C_VEL
LIN {X 0,Y 510.417,Z 584.641,A -85,B 0,C 180,E1 -5501.315,E2 -5501.315} C_VEL
LIN {X 0,Y 510.764,Z 573.786,A -85,B 0,C 180,E1 -5502.147,E2 -5502.147} C_VEL
LIN {X 0,Y 511.061,Z 562.9,A -85,B 0,C 180,E1 -5502.812,E2 -5502.812} C_VEL
LIN {X 0,Y 511.366,Z 551.217,A -85,B 0,C 180,E1 -5503.36,E2 -5503.36} C_VEL
LIN {X 0,Y 511.629,Z 537.751,A -85,B 0,C 180,E1 -5503.808,E2 -5503.808} C_VEL
LIN {X 0,Y 511.816,Z 524.382,A -85,B 0,C 180,E1 -5504.082,E2 -5504.082} C_VEL
LIN {X 0,Y 512.174,Z 434.413,A -85,B 0,C 180,E1 -5505.352,E2 -5505.352} C_VEL
LIN {X 0,Y 510.277,Z 422.838,A -85,B 0,C 180,E1 -5505.6,E2 -5505.6} C_VEL
LIN {X 0,Y 510.717,Z 406.754,A -85,B 0,C 180,E1 -5508.283,E2 -5508.283} C_VEL
LIN {X 0,Y 511.275,Z 387.641,A -85,B 0,C 180,E1 -5511.574,E2 -5511.574} C_VEL
LIN {X 0,Y 511.215,Z 382.791,A -85,B 0,C 180,E1 -5512.426,E2 -5512.426} C_VEL
LIN {X 0,Y 509.905,Z 375.57,A -85,B 0,C 180,E1 -5513.802,E2 -5513.802} C_VEL
LIN {X 0,Y 509.887,Z 375.471,A -85,B 0,C 180,E1 -5517.055,E2 -5517.055} C_VEL
LIN {X 0,Y 509.858,Z 375.475,A -85,B 0,C 180,E1 -5519.751,E2 -5519.751} C_VEL
LIN {X 0,Y 509.877,Z 375.469,A -85,B 0,C 180,E1 -5522.774,E2 -5522.774} C_VEL
LIN {X 0,Y 509.843,Z 375.478,A -85,B 0,C 180,E1 -5525.581,E2 -5525.581} C_VEL
LIN {X 0,Y 509.851,Z 375.472,A -85,B 0,C 180,E1 -5528.337,E2 -5528.337} C_VEL
LIN {X 0,Y 509.858,Z 375.477,A -85,B 0,C 180,E1 -5531.425,E2 -5531.425} C_VEL
LIN {X 0,Y 509.855,Z 375.473,A -85,B 0,C 180,E1 -5534.667,E2 -5534.667} C_VEL
LIN {X 0,Y 509.884,Z 375.468,A -85,B 0,C 180,E1 -5538.099,E2 -5538.099} C_VEL
LIN {X 0,Y 509.874,Z 375.472,A -85,B 0,C 180,E1 -5540.65,E2 -5540.65} C_VEL
LIN {X 0,Y 509.832,Z 375.476,A -85,B 0,C 180,E1 -5543.647,E2 -5543.647} C_VEL
LIN {X 0,Y 509.859,Z 375.474,A -85,B 0,C 180,E1 -5546.539,E2 -5546.539} C_VEL
LIN {X 0,Y 509.842,Z 375.477,A -85,B 0,C 180,E1 -5549.334,E2 -5549.334} C_VEL
LIN {X 0,Y 509.89,Z 375.468,A -85,B 0,C 180,E1 -5552.054,E2 -5552.054} C_VEL
LIN {X 0,Y 509.873,Z 375.474,A -85,B 0,C 180,E1 -5554.704,E2 -5554.704} C_VEL
LIN {X 0,Y 509.822,Z 375.477,A -85,B 0,C 180,E1 -5557.457,E2 -5557.457} C_VEL
LIN {X 0,Y 509.911,Z 375.465,A -85,B 0,C 180,E1 -5559.844,E2 -5559.844} C_VEL
LIN {X 0,Y 509.881,Z 375.472,A -85,B 0,C 180,E1 -5563.175,E2 -5563.175} C_VEL
LIN {X 0,Y 509.858,Z 375.472,A -85,B 0,C 180,E1 -5565.634,E2 -5565.634} C_VEL
LIN {X 0,Y 509.907,Z 375.471,A -85,B 0,C 180,E1 -5568.874,E2 -5568.874} C_VEL
LIN {X 0,Y 509.945,Z 375.464,A -85,B 0,C 180,E1 -5572.078,E2 -5572.078} C_VEL
LIN {X 0,Y 509.976,Z 375.462,A -85,B 0,C 180,E1 -5574.464,E2 -5574.464} C_VEL
LIN {X 0,Y 510.048,Z 375.449,A -85,B 0,C 180,E1 -5577.631,E2 -5577.631} C_VEL
LIN {X 0,Y 510.058,Z 375.451,A -85,B 0,C 180,E1 -5580.789,E2 -5580.789} C_VEL
LIN {X 0,Y 509.952,Z 375.461,A -85,B 0,C 180,E1 -5583.16,E2 -5583.16} C_VEL
LIN {X 0,Y 509.972,Z 375.462,A -85,B 0,C 180,E1 -5586.33,E2 -5586.33} C_VEL
LIN {X 0,Y 509.91,Z 375.468,A -85,B 0,C 180,E1 -5588.72,E2 -5588.72} C_VEL
LIN {X 0,Y 509.897,Z 375.472,A -85,B 0,C 180,E1 -5591.932,E2 -5591.932} C_VEL
LIN {X 0,Y 509.887,Z 375.469,A -85,B 0,C 180,E1 -5595.242,E2 -5595.242} C_VEL
LIN {X 0,Y 509.882,Z 375.474,A -85,B 0,C 180,E1 -5598.001,E2 -5598.001} C_VEL
LIN {X 0,Y 509.845,Z 375.474,A -85,B 0,C 180,E1 -5601.002,E2 -5601.002} C_VEL
LIN {X 0,Y 509.831,Z 375.479,A -85,B 0,C 180,E1 -5603.563,E2 -5603.563} C_VEL
LIN {X 0,Y 509.908,Z 375.469,A -85,B 0,C 180,E1 -5606.379,E2 -5606.379} C_VEL
LIN {X 0,Y 509.881,Z 375.469,A -85,B 0,C 180,E1 -5608.844,E2 -5608.844} C_VEL
LIN {X 0,Y 509.823,Z 375.482,A -85,B 0,C 180,E1 -5611.59,E2 -5611.59} C_VEL
LIN {X 0,Y 509.85,Z 375.474,A -85,B 0,C 180,E1 -5614.414,E2 -5614.414} C_VEL
LIN {X 0,Y 509.815,Z 375.481,A -85,B 0,C 180,E1 -5617.341,E2 -5617.341} C_VEL
LIN {X 0,Y 509.835,Z 375.475,A -85,B 0,C 180,E1 -5620.383,E2 -5620.383} C_VEL
LIN {X 0,Y 509.837,Z 375.476,A -85,B 0,C 180,E1 -5623.065,E2 -5623.065} C_VEL
LIN {X 0,Y 509.828,Z 375.479,A -85,B 0,C 180,E1 -5625.793,E2 -5625.793} C_VEL
LIN {X 0,Y 509.863,Z 375.471,A -85,B 0,C 180,E1 -5628.576,E2 -5628.576} C_VEL
LIN {X 0,Y 509.851,Z 375.475,A -85,B 0,C 180,E1 -5631.787,E2 -5631.787} C_VEL
LIN {X 0,Y 509.83,Z 375.478,A -85,B 0,C 180,E1 -5633.746,E2 -5633.746} C_VEL
LIN {X 0,Y 509.165,Z 375.558,A -85,B 0,C 180,E1 -5634.406,E2 -5634.406} C_VEL
LIN {X 0,Y 506.348,Z 375.914,A -85,B 0,C 180,E1 -5635.478,E2 -5635.478} C_VEL
LIN {X 0,Y 503.954,Z 376.212,A -85,B 0,C 180,E1 -5636.341,E2 -5636.341} C_VEL
LIN {X 0,Y 502.905,Z 376.341,A -85,B 0,C 180,E1 -5637.008,E2 -5637.008} C_VEL
LIN {X 0,Y 502.807,Z 376.351,A -85,B 0,C 180,E1 -5637.233,E2 -5637.233} C_VEL
LIN {X 0,Y 502.815,Z 376.349,A -85,B 0,C 180,E1 -5640.065,E2 -5640.065} C_VEL
LIN {X 0,Y 502.833,Z 376.347,A -85,B 0,C 180,E1 -5642.534,E2 -5642.534} C_VEL
LIN {X 0,Y 502.827,Z 376.352,A -85,B 0,C 180,E1 -5645.299,E2 -5645.299} C_VEL
LIN {X 0,Y 502.781,Z 376.353,A -85,B 0,C 180,E1 -5647.827,E2 -5647.827} C_VEL
LIN {X 0,Y 502.825,Z 376.347,A -85,B 0,C 180,E1 -5650.4,E2 -5650.4} C_VEL
LIN {X 0,Y 502.832,Z 376.353,A -85,B 0,C 180,E1 -5652.932,E2 -5652.932} C_VEL
LIN {X 0,Y 502.847,Z 376.348,A -85,B 0,C 180,E1 -5655.429,E2 -5655.429} C_VEL
LIN {X 0,Y 502.88,Z 376.347,A -85,B 0,C 180,E1 -5658.717,E2 -5658.717} C_VEL
LIN {X 0,Y 502.952,Z 376.548,A -85,B 0,C 180,E1 -5660.905,E2 -5660.905} C_VEL
LIN {X 0,Y 503.998,Z 383.199,A -85,B 0,C 180,E1 -5662.258,E2 -5662.258} C_VEL
LIN {X 0,Y 503.73,Z 393.309,A -85,B 0,C 180,E1 -5664.194,E2 -5664.194} C_VEL
LIN {X 0,Y 503.313,Z 409.324,A -85,B 0,C 180,E1 -5667.199,E2 -5667.199} C_VEL
LIN {X 0,Y 503.554,Z 411.19,A -85,B 0,C 180,E1 -5667.287,E2 -5667.287} C_VEL
LIN {X 0,Y 505.469,Z 422.214,A -85,B 0,C 180,E1 -5667.51,E2 -5667.51} C_VEL
LIN {X 0,Y 504.861,Z 516.752,A -85,B 0,C 180,E1 -5668.878,E2 -5668.878} C_VEL
LIN {X 0,Y 504.635,Z 530.526,A -85,B 0,C 180,E1 -5669.252,E2 -5669.252} C_VEL
LIN {X 0,Y 504.362,Z 542.881,A -85,B 0,C 180,E1 -5669.75,E2 -5669.75} C_VEL
LIN {X 0,Y 503.966,Z 554.745,A -85,B 0,C 180,E1 -5670.399,E2 -5670.399} C_VEL
LIN {X 0,Y 503.548,Z 566.102,A -85,B 0,C 180,E1 -5671.199,E2 -5671.199} C_VEL
LIN {X 0,Y 503.239,Z 576.333,A -85,B 0,C 180,E1 -5672.101,E2 -5672.101} C_VEL
LIN {X 0,Y 502.929,Z 584.74,A -85,B 0,C 180,E1 -5673.004,E2 -5673.004} C_VEL
LIN {X 0,Y 502.657,Z 593.866,A -85,B 0,C 180,E1 -5674.209,E2 -5674.209} C_VEL
LIN {X 0,Y 502.362,Z 601.244,A -85,B 0,C 180,E1 -5675.418,E2 -5675.418} C_VEL
LIN {X 0,Y 502.29,Z 608.034,A -85,B 0,C 180,E1 -5676.83,E2 -5676.83} C_VEL
LIN {X 0,Y 502.187,Z 612.537,A -85,B 0,C 180,E1 -5678.044,E2 -5678.044} C_VEL
LIN {X 0,Y 502.117,Z 614.918,A -85,B 0,C 180,E1 -5678.856,E2 -5678.856} C_VEL
LIN {X 0,Y 502.036,Z 616.872,A -85,B 0,C 180,E1 -5679.67,E2 -5679.67} C_VEL
LIN {X 0,Y 502.046,Z 618.395,A -85,B 0,C 180,E1 -5680.485,E2 -5680.485} C_VEL
LIN {X 0,Y 502.09,Z 619.684,A -85,B 0,C 180,E1 -5681.528,E2 -5681.528} C_VEL
LIN {X 0,Y 501.981,Z 620.401,A -85,B 0,C 180,E1 -5682.944,E2 -5682.944} C_VEL
LIN {X 0,Y 502.002,Z 620.248,A -85,B 0,C 180,E1 -5683.768,E2 -5683.768} C_VEL
LIN {X 0,Y 502.022,Z 619.249,A -85,B 0,C 180,E1 -5684.993,E2 -5684.993} C_VEL
LIN {X 0,Y 502.015,Z 617.223,A -85,B 0,C 180,E1 -5686.259,E2 -5686.259} C_VEL
LIN {X 0,Y 502.126,Z 614.257,A -85,B 0,C 180,E1 -5687.485,E2 -5687.485} C_VEL
LIN {X 0,Y 502.217,Z 609.986,A -85,B 0,C 180,E1 -5688.775,E2 -5688.775} C_VEL
LIN {X 0,Y 502.325,Z 604.644,A -85,B 0,C 180,E1 -5690.013,E2 -5690.013} C_VEL
LIN {X 0,Y 502.564,Z 597.492,A -85,B 0,C 180,E1 -5691.32,E2 -5691.32} C_VEL
LIN {X 0,Y 502.803,Z 589.795,A -85,B 0,C 180,E1 -5692.453,E2 -5692.453} C_VEL
LIN {X 0,Y 503.11,Z 580.444,A -85,B 0,C 180,E1 -5693.569,E2 -5693.569} C_VEL
LIN {X 0,Y 503.466,Z 570.374,A -85,B 0,C 180,E1 -5694.537,E2 -5694.537} C_VEL
LIN {X 0,Y 503.859,Z 559.105,A -85,B 0,C 180,E1 -5695.408,E2 -5695.408} C_VEL
LIN {X 0,Y 504.187,Z 546.596,A -85,B 0,C 180,E1 -5696.156,E2 -5696.156} C_VEL
LIN {X 0,Y 504.561,Z 534.812,A -85,B 0,C 180,E1 -5696.684,E2 -5696.684} C_VEL
LIN {X 0,Y 504.782,Z 521.487,A -85,B 0,C 180,E1 -5697.107,E2 -5697.107} C_VEL
LIN {X 0,Y 504.943,Z 507.081,A -85,B 0,C 180,E1 -5697.37,E2 -5697.37} C_VEL
LIN {X 0,Y 505.309,Z 421.076,A -85,B 0,C 180,E1 -5698.602,E2 -5698.602} C_VEL
LIN {X 0,Y 503.32,Z 409.753,A -85,B 0,C 180,E1 -5698.853,E2 -5698.853} C_VEL
LIN {X 0,Y 503.384,Z 406.087,A -85,B 0,C 180,E1 -5699.481,E2 -5699.481} C_VEL
LIN {X 0,Y 503.927,Z 389.101,A -85,B 0,C 180,E1 -5702.712,E2 -5702.712} C_VEL
LIN {X 0,Y 504.038,Z 382.975,A -85,B 0,C 180,E1 -5703.898,E2 -5703.898} C_VEL
LIN {X 0,Y 502.812,Z 376.401,A -85,B 0,C 180,E1 -5705.3,E2 -5705.3} C_VEL
LIN {X 0,Y 502.805,Z 376.352,A -85,B 0,C 180,E1 -5708.487,E2 -5708.487} C_VEL
LIN {X 0,Y 502.823,Z 376.353,A -85,B 0,C 180,E1 -5711.064,E2 -5711.064} C_VEL
LIN {X 0,Y 502.777,Z 376.359,A -85,B 0,C 180,E1 -5713.375,E2 -5713.375} C_VEL
LIN {X 0,Y 502.785,Z 376.354,A -85,B 0,C 180,E1 -5715.661,E2 -5715.661} C_VEL
LIN {X 0,Y 502.834,Z 376.343,A -85,B 0,C 180,E1 -5717.865,E2 -5717.865} C_VEL
LIN {X 0,Y 502.816,Z 376.351,A -85,B 0,C 180,E1 -5721.025,E2 -5721.025} C_VEL
LIN {X 0,Y 502.78,Z 376.352,A -85,B 0,C 180,E1 -5724.166,E2 -5724.166} C_VEL
LIN {X 0,Y 502.826,Z 376.352,A -85,B 0,C 180,E1 -5726.993,E2 -5726.993} C_VEL
LIN {X 0,Y 502.823,Z 376.34,A -85,B 0,C 180,E1 -5730.061,E2 -5730.061} C_VEL
LIN {X 0,Y 502.828,Z 376.348,A -85,B 0,C 180,E1 -5732.533,E2 -5732.533} C_VEL
LIN {X 0,Y 502.823,Z 376.352,A -85,B 0,C 180,E1 -5735.297,E2 -5735.297} C_VEL
LIN {X 0,Y 502.802,Z 376.347,A -85,B 0,C 180,E1 -5737.827,E2 -5737.827} C_VEL
LIN {X 0,Y 502.818,Z 376.349,A -85,B 0,C 180,E1 -5740.4,E2 -5740.4} C_VEL
LIN {X 0,Y 502.828,Z 376.353,A -85,B 0,C 180,E1 -5742.931,E2 -5742.931} C_VEL
LIN {X 0,Y 502.836,Z 376.345,A -85,B 0,C 180,E1 -5745.429,E2 -5745.429} C_VEL
LIN {X 0,Y 502.886,Z 376.345,A -85,B 0,C 180,E1 -5748.717,E2 -5748.717} C_VEL
LIN {X 0,Y 502.893,Z 376.338,A -85,B 0,C 180,E1 -5751.967,E2 -5751.967} C_VEL
LIN {X 0,Y 502.939,Z 376.332,A -85,B 0,C 180,E1 -5754.387,E2 -5754.387} C_VEL
LIN {X 0,Y 503.019,Z 376.322,A -85,B 0,C 180,E1 -5757.598,E2 -5757.598} C_VEL
LIN {X 0,Y 503.017,Z 376.321,A -85,B 0,C 180,E1 -5760,E2 -5760} C_VEL
LIN {X 0,Y 503.017,Z 376.326,A -85,B 0,C 180,E1 -5762.402,E2 -5762.402} C_VEL
LIN {X 0,Y 502.939,Z 376.332,A -85,B 0,C 180,E1 -5765.614,E2 -5765.614} C_VEL
LIN {X 0,Y 502.893,Z 376.337,A -85,B 0,C 180,E1 -5768.034,E2 -5768.034} C_VEL
LIN {X 0,Y 502.886,Z 376.341,A -85,B 0,C 180,E1 -5771.283,E2 -5771.283} C_VEL
LIN {X 0,Y 502.836,Z 376.347,A -85,B 0,C 180,E1 -5774.571,E2 -5774.571} C_VEL
LIN {X 0,Y 502.853,Z 376.341,A -85,B 0,C 180,E1 -5777.907,E2 -5777.907} C_VEL
LIN {X 0,Y 502.822,Z 376.353,A -85,B 0,C 180,E1 -5780.537,E2 -5780.537} C_VEL
LIN {X 0,Y 502.798,Z 376.352,A -85,B 0,C 180,E1 -5783.04,E2 -5783.04} C_VEL
LIN {X 0,Y 502.834,Z 376.344,A -85,B 0,C 180,E1 -5785.676,E2 -5785.676} C_VEL
LIN {X 0,Y 502.833,Z 376.349,A -85,B 0,C 180,E1 -5788.373,E2 -5788.373} C_VEL
LIN {X 0,Y 502.789,Z 376.351,A -85,B 0,C 180,E1 -5791.5,E2 -5791.5} C_VEL
LIN {X 0,Y 502.801,Z 376.354,A -85,B 0,C 180,E1 -5794.446,E2 -5794.446} C_VEL
LIN {X 0,Y 502.776,Z 376.353,A -85,B 0,C 180,E1 -5797.179,E2 -5797.179} C_VEL
LIN {X 0,Y 502.817,Z 376.349,A -85,B 0,C 180,E1 -5800.013,E2 -5800.013} C_VEL
LIN {X 0,Y 502.825,Z 376.343,A -85,B 0,C 180,E1 -5802.203,E2 -5802.203} C_VEL
LIN {X 0,Y 502.796,Z 376.348,A -85,B 0,C 180,E1 -5805.469,E2 -5805.469} C_VEL
LIN {X 0,Y 502.826,Z 376.347,A -85,B 0,C 180,E1 -5807.865,E2 -5807.865} C_VEL
LIN {X 0,Y 502.8,Z 376.353,A -85,B 0,C 180,E1 -5811.025,E2 -5811.025} C_VEL
LIN {X 0,Y 502.784,Z 376.353,A -85,B 0,C 180,E1 -5814.168,E2 -5814.168} C_VEL
LIN {X 0,Y 502.832,Z 376.349,A -85,B 0,C 180,E1 -5816.994,E2 -5816.994} C_VEL
LIN {X 0,Y 502.814,Z 376.354,A -85,B 0,C 180,E1 -5820.066,E2 -5820.066} C_VEL
LIN {X 0,Y 502.835,Z 376.353,A -85,B 0,C 180,E1 -5822.534,E2 -5822.534} C_VEL
LIN {X 0,Y 502.849,Z 376.351,A -85,B 0,C 180,E1 -5825.651,E2 -5825.651} C_VEL
LIN {X 0,Y 502.888,Z 376.567,A -85,B 0,C 180,E1 -5826.037,E2 -5826.037} C_VEL
LIN {X 0,Y 504.376,Z 385.189,A -85,B 0,C 180,E1 -5827.685,E2 -5827.685} C_VEL
LIN {X 0,Y 503.96,Z 398.422,A -85,B 0,C 180,E1 -5830.022,E2 -5830.022} C_VEL
LIN {X 0,Y 503.5,Z 414.122,A -85,B 0,C 180,E1 -5832.746,E2 -5832.746} C_VEL
LIN {X 0,Y 503.278,Z 422.673,A -85,B 0,C 180,E1 -5834.174,E2 -5834.174} C_VEL
LIN {X 0,Y 505.389,Z 435.572,A -85,B 0,C 180,E1 -5834.456,E2 -5834.456} C_VEL
LIN {X 0,Y 504.903,Z 530.163,A -85,B 0,C 180,E1 -5835.825,E2 -5835.825} C_VEL
LIN {X 0,Y 504.592,Z 543.505,A -85,B 0,C 180,E1 -5836.176,E2 -5836.176} C_VEL
LIN {X 0,Y 504.286,Z 556.827,A -85,B 0,C 180,E1 -5836.706,E2 -5836.706} C_VEL
LIN {X 0,Y 503.948,Z 568.848,A -85,B 0,C 180,E1 -5837.367,E2 -5837.367} C_VEL
LIN {X 0,Y 503.582,Z 580.898,A -85,B 0,C 180,E1 -5838.223,E2 -5838.223} C_VEL
LIN {X 0,Y 503.207,Z 591.093,A -85,B 0,C 180,E1 -5839.132,E2 -5839.132} C_VEL
LIN {X 0,Y 502.884,Z 600.262,A -85,B 0,C 180,E1 -5840.143,E2 -5840.143} C_VEL
LIN {X 0,Y 502.618,Z 609.193,A -85,B 0,C 180,E1 -5841.355,E2 -5841.355} C_VEL
LIN {X 0,Y 502.36,Z 616.379,A -85,B 0,C 180,E1 -5842.565,E2 -5842.565} C_VEL
LIN {X 0,Y 502.235,Z 621.229,A -85,B 0,C 180,E1 -5843.573,E2 -5843.573} C_VEL
LIN {X 0,Y 502.181,Z 625.942,A -85,B 0,C 180,E1 -5844.781,E2 -5844.781} C_VEL
LIN {X 0,Y 502.139,Z 629.541,A -85,B 0,C 180,E1 -5845.987,E2 -5845.987} C_VEL
LIN {X 0,Y 502.12,Z 631.398,A -85,B 0,C 180,E1 -5846.791,E2 -5846.791} C_VEL
LIN {X 0,Y 502.035,Z 633.783,A -85,B 0,C 180,E1 -5848.396,E2 -5848.396} C_VEL
LIN {X 0,Y 501.98,Z 634.605,A -85,B 0,C 180,E1 -5850,E2 -5850} C_VEL
LIN {X 0,Y 502.035,Z 633.787,A -85,B 0,C 180,E1 -5851.605,E2 -5851.605} C_VEL
LIN {X 0,Y 502.12,Z 631.406,A -85,B 0,C 180,E1 -5853.21,E2 -5853.21} C_VEL
LIN {X 0,Y 502.104,Z 628.479,A -85,B 0,C 180,E1 -5854.415,E2 -5854.415} C_VEL
LIN {X 0,Y 502.235,Z 624.518,A -85,B 0,C 180,E1 -5855.621,E2 -5855.621} C_VEL
LIN {X 0,Y 502.333,Z 618.524,A -85,B 0,C 180,E1 -5857.012,E2 -5857.012} C_VEL
LIN {X 0,Y 502.498,Z 611.76,A -85,B 0,C 180,E1 -5858.242,E2 -5858.242} C_VEL
LIN {X 0,Y 502.763,Z 603.492,A -85,B 0,C 180,E1 -5859.454,E2 -5859.454} C_VEL
LIN {X 0,Y 503.046,Z 595.012,A -85,B 0,C 180,E1 -5860.464,E2 -5860.464} C_VEL
LIN {X 0,Y 503.433,Z 584.532,A -85,B 0,C 180,E1 -5861.474,E2 -5861.474} C_VEL
LIN {X 0,Y 503.783,Z 573.674,A -85,B 0,C 180,E1 -5862.318,E2 -5862.318} C_VEL
LIN {X 0,Y 504.119,Z 562.785,A -85,B 0,C 180,E1 -5862.991,E2 -5862.991} C_VEL
LIN {X 0,Y 504.457,Z 551.096,A -85,B 0,C 180,E1 -5863.546,E2 -5863.546} C_VEL
LIN {X 0,Y 504.739,Z 537.622,A -85,B 0,C 180,E1 -5864,E2 -5864} C_VEL
LIN {X 0,Y 504.938,Z 524.227,A -85,B 0,C 180,E1 -5864.277,E2 -5864.277} C_VEL
LIN {X 0,Y 505.257,Z 434.489,A -85,B 0,C 180,E1 -5865.564,E2 -5865.564} C_VEL
LIN {X 0,Y 503.285,Z 422.707,A -85,B 0,C 180,E1 -5865.825,E2 -5865.825} C_VEL
LIN {X 0,Y 503.751,Z 407.316,A -85,B 0,C 180,E1 -5868.433,E2 -5868.433} C_VEL
LIN {X 0,Y 504.372,Z 387.533,A -85,B 0,C 180,E1 -5871.884,E2 -5871.884} C_VEL
LIN {X 0,Y 504.218,Z 383.887,A -85,B 0,C 180,E1 -5872.538,E2 -5872.538} C_VEL
LIN {X 0,Y 502.857,Z 376.476,A -85,B 0,C 180,E1 -5873.965,E2 -5873.965} C_VEL
LIN {X 0,Y 502.865,Z 376.343,A -85,B 0,C 180,E1 -5876.566,E2 -5876.566} C_VEL
LIN {X 0,Y 502.825,Z 376.354,A -85,B 0,C 180,E1 -5879.287,E2 -5879.287} C_VEL
LIN {X 0,Y 502.789,Z 376.352,A -85,B 0,C 180,E1 -5882.084,E2 -5882.084} C_VEL
LIN {X 0,Y 502.81,Z 376.351,A -85,B 0,C 180,E1 -5884.964,E2 -5884.964} C_VEL
LIN {X 0,Y 502.795,Z 376.352,A -85,B 0,C 180,E1 -5887.953,E2 -5887.953} C_VEL
LIN {X 0,Y 502.82,Z 376.352,A -85,B 0,C 180,E1 -5891.065,E2 -5891.065} C_VEL
LIN {X 0,Y 502.788,Z 376.352,A -85,B 0,C 180,E1 -5894.338,E2 -5894.338} C_VEL
LIN {X 0,Y 502.785,Z 376.355,A -85,B 0,C 180,E1 -5896.77,E2 -5896.77} C_VEL
LIN {X 0,Y 502.826,Z 376.352,A -85,B 0,C 180,E1 -5899.003,E2 -5899.003} C_VEL
LIN {X 0,Y 502.794,Z 376.352,A -85,B 0,C 180,E1 -5902.046,E2 -5902.046} C_VEL
LIN {X 0,Y 502.806,Z 376.356,A -85,B 0,C 180,E1 -5905.035,E2 -5905.035} C_VEL
LIN {X 0,Y 502.783,Z 376.353,A -85,B 0,C 180,E1 -5907.915,E2 -5907.915} C_VEL
LIN {X 0,Y 502.82,Z 376.352,A -85,B 0,C 180,E1 -5910.712,E2 -5910.712} C_VEL
LIN {X 0,Y 502.876,Z 376.343,A -85,B 0,C 180,E1 -5913.434,E2 -5913.434} C_VEL
LIN {X 0,Y 502.786,Z 376.354,A -85,B 0,C 180,E1 -5916.086,E2 -5916.086} C_VEL
LIN {X 0,Y 502.778,Z 376.358,A -85,B 0,C 180,E1 -5918.688,E2 -5918.688} C_VEL
LIN {X 0,Y 502.825,Z 376.35,A -85,B 0,C 180,E1 -5921.248,E2 -5921.248} C_VEL
LIN {X 0,Y 502.818,Z 376.349,A -85,B 0,C 180,E1 -5923.767,E2 -5923.767} C_VEL
LIN {X 0,Y 502.825,Z 376.352,A -85,B 0,C 180,E1 -5926.254,E2 -5926.254} C_VEL
LIN {X 0,Y 502.871,Z 376.347,A -85,B 0,C 180,E1 -5928.717,E2 -5928.717} C_VEL
LIN {X 0,Y 502.895,Z 376.342,A -85,B 0,C 180,E1 -5931.966,E2 -5931.966} C_VEL
LIN {X 0,Y 502.932,Z 376.339,A -85,B 0,C 180,E1 -5934.386,E2 -5934.386} C_VEL
LIN {X 0,Y 503.018,Z 376.325,A -85,B 0,C 180,E1 -5937.598,E2 -5937.598} C_VEL
LIN {X 0,Y 503.02,Z 376.328,A -85,B 0,C 180,E1 -5940,E2 -5940} C_VEL
LIN {X 0,Y 503.018,Z 376.328,A -85,B 0,C 180,E1 -5942.402,E2 -5942.402} C_VEL
LIN {X 0,Y 502.933,Z 376.336,A -85,B 0,C 180,E1 -5945.613,E2 -5945.613} C_VEL
LIN {X 0,Y 502.895,Z 376.344,A -85,B 0,C 180,E1 -5948.033,E2 -5948.033} C_VEL
LIN {X 0,Y 502.87,Z 376.343,A -85,B 0,C 180,E1 -5951.283,E2 -5951.283} C_VEL
LIN {X 0,Y 502.839,Z 376.35,A -85,B 0,C 180,E1 -5954.571,E2 -5954.571} C_VEL
LIN {X 0,Y 502.856,Z 376.349,A -85,B 0,C 180,E1 -5957.907,E2 -5957.907} C_VEL
LIN {X 0,Y 502.823,Z 376.351,A -85,B 0,C 180,E1 -5960.536,E2 -5960.536} C_VEL
LIN {X 0,Y 502.791,Z 376.353,A -85,B 0,C 180,E1 -5963.041,E2 -5963.041} C_VEL
LIN {X 0,Y 502.836,Z 376.352,A -85,B 0,C 180,E1 -5965.676,E2 -5965.676} C_VEL
LIN {X 0,Y 502.838,Z 376.349,A -85,B 0,C 180,E1 -5968.373,E2 -5968.373} C_VEL
LIN {X 0,Y 502.793,Z 376.357,A -85,B 0,C 180,E1 -5971.5,E2 -5971.5} C_VEL
LIN {X 0,Y 502.803,Z 376.352,A -85,B 0,C 180,E1 -5974.445,E2 -5974.445} C_VEL
LIN {X 0,Y 502.777,Z 376.356,A -85,B 0,C 180,E1 -5977.179,E2 -5977.179} C_VEL
LIN {X 0,Y 502.785,Z 376.356,A -85,B 0,C 180,E1 -5980.016,E2 -5980.016} C_VEL
LIN {X 0,Y 502.8,Z 376.353,A -85,B 0,C 180,E1 -5982.2,E2 -5982.2} C_VEL
LIN {X 0,Y 502.798,Z 376.357,A -85,B 0,C 180,E1 -5985.469,E2 -5985.469} C_VEL
LIN {X 0,Y 502.825,Z 376.35,A -85,B 0,C 180,E1 -5989.004,E2 -5989.004} C_VEL
LIN {X 0,Y 502.793,Z 376.353,A -85,B 0,C 180,E1 -5992.047,E2 -5992.047} C_VEL
LIN {X 0,Y 502.809,Z 376.353,A -85,B 0,C 180,E1 -5995.036,E2 -5995.036} C_VEL
LIN {X 0,Y 502.807,Z 376.351,A -85,B 0,C 180,E1 -5997.233,E2 -5997.233} C_VEL
LIN {X 0,Y 502.106,Z 376.439,A -85,B 0,C 180,E1 -5997.902,E2 -5997.902} C_VEL
LIN {X 0,Y 499.241,Z 376.798,A -85,B 0,C 180,E1 -5998.988,E2 -5998.988} C_VEL
LIN {X 0,Y 496.847,Z 377.094,A -85,B 0,C 180,E1 -5999.863,E2 -5999.863} C_VEL
LIN {X 0,Y 495.831,Z 377.219,A -85,B 0,C 180,E1 -6000.538,E2 -6000.538} C_VEL
LIN {X 0,Y 495.753,Z 377.23,A -85,B 0,C 180,E1 -6000.767,E2 -6000.767} C_VEL
LIN {X 0,Y 495.791,Z 377.224,A -85,B 0,C 180,E1 -6003.933,E2 -6003.933} C_VEL
LIN {X 0,Y 495.761,Z 377.234,A -85,B 0,C 180,E1 -6007.14,E2 -6007.14} C_VEL
LIN {X 0,Y 495.772,Z 377.225,A -85,B 0,C 180,E1 -6010.11,E2 -6010.11} C_VEL
LIN {X 0,Y 495.783,Z 377.227,A -85,B 0,C 180,E1 -6012.681,E2 -6012.681} C_VEL
LIN {X 0,Y 495.792,Z 377.23,A -85,B 0,C 180,E1 -6015.217,E2 -6015.217} C_VEL
LIN {X 0,Y 495.854,Z 377.221,A -85,B 0,C 180,E1 -6018.555,E2 -6018.555} C_VEL
LIN {X 0,Y 495.881,Z 377.367,A -85,B 0,C 180,E1 -6020.723,E2 -6020.723} C_VEL
LIN {X 0,Y 497.042,Z 384.302,A -85,B 0,C 180,E1 -6022.162,E2 -6022.162} C_VEL
LIN {X 0,Y 496.736,Z 394.367,A -85,B 0,C 180,E1 -6024.112,E2 -6024.112} C_VEL
LIN {X 0,Y 496.336,Z 409.517,A -85,B 0,C 180,E1 -6026.981,E2 -6026.981} C_VEL
LIN {X 0,Y 496.806,Z 412.576,A -85,B 0,C 180,E1 -6027.089,E2 -6027.089} C_VEL
LIN {X 0,Y 498.639,Z 422.803,A -85,B 0,C 180,E1 -6027.299,E2 -6027.299} C_VEL
LIN {X 0,Y 497.991,Z 517.129,A -85,B 0,C 180,E1 -6028.686,E2 -6028.686} C_VEL
LIN {X 0,Y 497.761,Z 530.803,A -85,B 0,C 180,E1 -6029.064,E2 -6029.064} C_VEL
LIN {X 0,Y 497.422,Z 543.645,A -85,B 0,C 180,E1 -6029.595,E2 -6029.595} C_VEL
LIN {X 0,Y 497.005,Z 556.114,A -85,B 0,C 180,E1 -6030.304,E2 -6030.304} C_VEL
LIN {X 0,Y 496.572,Z 567.239,A -85,B 0,C 180,E1 -6031.115,E2 -6031.115} C_VEL
LIN {X 0,Y 496.217,Z 577.272,A -85,B 0,C 180,E1 -6032.029,E2 -6032.029} C_VEL
LIN {X 0,Y 495.86,Z 586.343,A -85,B 0,C 180,E1 -6033.046,E2 -6033.046} C_VEL
LIN {X 0,Y 495.589,Z 595.191,A -85,B 0,C 180,E1 -6034.269,E2 -6034.269} C_VEL
LIN {X 0,Y 495.294,Z 602.353,A -85,B 0,C 180,E1 -6035.496,E2 -6035.496} C_VEL
LIN {X 0,Y 495.253,Z 607.581,A -85,B 0,C 180,E1 -6036.61,E2 -6036.61} C_VEL
LIN {X 0,Y 495.112,Z 611.893,A -85,B 0,C 180,E1 -6037.75,E2 -6037.75} C_VEL
LIN {X 0,Y 495.013,Z 615.508,A -85,B 0,C 180,E1 -6038.984,E2 -6038.984} C_VEL
LIN {X 0,Y 494.954,Z 617.369,A -85,B 0,C 180,E1 -6039.81,E2 -6039.81} C_VEL
LIN {X 0,Y 494.949,Z 618.757,A -85,B 0,C 180,E1 -6040.637,E2 -6040.637} C_VEL
LIN {X 0,Y 495.006,Z 619.854,A -85,B 0,C 180,E1 -6041.579,E2 -6041.579} C_VEL
LIN {X 0,Y 494.907,Z 620.504,A -85,B 0,C 180,E1 -6043.132,E2 -6043.132} C_VEL
LIN {X 0,Y 494.911,Z 620.236,A -85,B 0,C 180,E1 -6043.969,E2 -6043.969} C_VEL
LIN {X 0,Y 494.939,Z 619.278,A -85,B 0,C 180,E1 -6045.076,E2 -6045.076} C_VEL
LIN {X 0,Y 494.933,Z 616.908,A -85,B 0,C 180,E1 -6046.498,E2 -6046.498} C_VEL
LIN {X 0,Y 495.076,Z 613.037,A -85,B 0,C 180,E1 -6047.988,E2 -6047.988} C_VEL
LIN {X 0,Y 495.202,Z 607.589,A -85,B 0,C 180,E1 -6049.482,E2 -6049.482} C_VEL
LIN {X 0,Y 495.383,Z 601.39,A -85,B 0,C 180,E1 -6050.773,E2 -6050.773} C_VEL
LIN {X 0,Y 495.652,Z 593.56,A -85,B 0,C 180,E1 -6052.07,E2 -6052.07} C_VEL
LIN {X 0,Y 495.974,Z 584.95,A -85,B 0,C 180,E1 -6053.217,E2 -6053.217} C_VEL
LIN {X 0,Y 496.297,Z 575.395,A -85,B 0,C 180,E1 -6054.246,E2 -6054.246} C_VEL
LIN {X 0,Y 496.716,Z 564.066,A -85,B 0,C 180,E1 -6055.228,E2 -6055.228} C_VEL
LIN {X 0,Y 497.145,Z 552.895,A -85,B 0,C 180,E1 -6055.991,E2 -6055.991} C_VEL
LIN {X 0,Y 497.495,Z 541.583,A -85,B 0,C 180,E1 -6056.592,E2 -6056.592} C_VEL
LIN {X 0,Y 497.808,Z 528.16,A -85,B 0,C 180,E1 -6057.116,E2 -6057.116} C_VEL
LIN {X 0,Y 498.038,Z 515.879,A -85,B 0,C 180,E1 -6057.43,E2 -6057.43} C_VEL
LIN {X 0,Y 498.539,Z 422.205,A -85,B 0,C 180,E1 -6058.806,E2 -6058.806} C_VEL
LIN {X 0,Y 496.385,Z 410.128,A -85,B 0,C 180,E1 -6059.073,E2 -6059.073} C_VEL
LIN {X 0,Y 496.348,Z 408.719,A -85,B 0,C 180,E1 -6059.242,E2 -6059.242} C_VEL
LIN {X 0,Y 496.912,Z 391.737,A -85,B 0,C 180,E1 -6062.509,E2 -6062.509} C_VEL
LIN {X 0,Y 497.113,Z 384.396,A -85,B 0,C 180,E1 -6063.946,E2 -6063.946} C_VEL
LIN {X 0,Y 495.758,Z 377.284,A -85,B 0,C 180,E1 -6065.486,E2 -6065.486} C_VEL
LIN {X 0,Y 495.775,Z 377.23,A -85,B 0,C 180,E1 -6068.77,E2 -6068.77} C_VEL
LIN {X 0,Y 495.775,Z 377.228,A -85,B 0,C 180,E1 -6071.778,E2 -6071.778} C_VEL
LIN {X 0,Y 495.744,Z 377.233,A -85,B 0,C 180,E1 -6075.139,E2 -6075.139} C_VEL
LIN {X 0,Y 495.78,Z 377.221,A -85,B 0,C 180,E1 -6078.221,E2 -6078.221} C_VEL
LIN {X 0,Y 495.773,Z 377.228,A -85,B 0,C 180,E1 -6081.229,E2 -6081.229} C_VEL
LIN {X 0,Y 495.752,Z 377.229,A -85,B 0,C 180,E1 -6084.463,E2 -6084.463} C_VEL
LIN {X 0,Y 495.762,Z 377.231,A -85,B 0,C 180,E1 -6087.405,E2 -6087.405} C_VEL
LIN {X 0,Y 495.774,Z 377.219,A -85,B 0,C 180,E1 -6090.254,E2 -6090.254} C_VEL
LIN {X 0,Y 495.826,Z 377.224,A -85,B 0,C 180,E1 -6093.248,E2 -6093.248} C_VEL
LIN {X 0,Y 495.75,Z 377.229,A -85,B 0,C 180,E1 -6095.725,E2 -6095.725} C_VEL
LIN {X 0,Y 495.752,Z 377.226,A -85,B 0,C 180,E1 -6098.371,E2 -6098.371} C_VEL
LIN {X 0,Y 495.777,Z 377.23,A -85,B 0,C 180,E1 -6100.971,E2 -6100.971} C_VEL
LIN {X 0,Y 495.772,Z 377.227,A -85,B 0,C 180,E1 -6103.53,E2 -6103.53} C_VEL
LIN {X 0,Y 495.788,Z 377.221,A -85,B 0,C 180,E1 -6106.056,E2 -6106.056} C_VEL
LIN {X 0,Y 495.866,Z 377.217,A -85,B 0,C 180,E1 -6108.555,E2 -6108.555} C_VEL
LIN {X 0,Y 495.864,Z 377.214,A -85,B 0,C 180,E1 -6111.852,E2 -6111.852} C_VEL
LIN {X 0,Y 495.895,Z 377.209,A -85,B 0,C 180,E1 -6114.307,E2 -6114.307} C_VEL
LIN {X 0,Y 495.989,Z 377.198,A -85,B 0,C 180,E1 -6117.564,E2 -6117.564} C_VEL
LIN {X 0,Y 495.988,Z 377.196,A -85,B 0,C 180,E1 -6120,E2 -6120} C_VEL
LIN {X 0,Y 495.986,Z 377.202,A -85,B 0,C 180,E1 -6122.436,E2 -6122.436} C_VEL
LIN {X 0,Y 495.895,Z 377.209,A -85,B 0,C 180,E1 -6125.694,E2 -6125.694} C_VEL
LIN {X 0,Y 495.864,Z 377.213,A -85,B 0,C 180,E1 -6128.148,E2 -6128.148} C_VEL
LIN {X 0,Y 495.86,Z 377.215,A -85,B 0,C 180,E1 -6131.445,E2 -6131.445} C_VEL
LIN {X 0,Y 495.781,Z 377.23,A -85,B 0,C 180,E1 -6134.783,E2 -6134.783} C_VEL
LIN {X 0,Y 495.78,Z 377.223,A -85,B 0,C 180,E1 -6137.319,E2 -6137.319} C_VEL
LIN {X 0,Y 495.77,Z 377.225,A -85,B 0,C 180,E1 -6139.891,E2 -6139.891} C_VEL
LIN {X 0,Y 495.757,Z 377.231,A -85,B 0,C 180,E1 -6142.863,E2 -6142.863} C_VEL
LIN {X 0,Y 495.792,Z 377.223,A -85,B 0,C 180,E1 -6146.068,E2 -6146.068} C_VEL
LIN {X 0,Y 495.765,Z 377.232,A -85,B 0,C 180,E1 -6148.815,E2 -6148.815} C_VEL
LIN {X 0,Y 495.752,Z 377.227,A -85,B 0,C 180,E1 -6151.727,E2 -6151.727} C_VEL
LIN {X 0,Y 495.771,Z 377.232,A -85,B 0,C 180,E1 -6154.696,E2 -6154.696} C_VEL
LIN {X 0,Y 495.726,Z 377.229,A -85,B 0,C 180,E1 -6157.562,E2 -6157.562} C_VEL
LIN {X 0,Y 495.775,Z 377.223,A -85,B 0,C 180,E1 -6160.699,E2 -6160.699} C_VEL
LIN {X 0,Y 495.73,Z 377.231,A -85,B 0,C 180,E1 -6163.696,E2 -6163.696} C_VEL
LIN {X 0,Y 495.731,Z 377.232,A -85,B 0,C 180,E1 -6166.305,E2 -6166.305} C_VEL
LIN {X 0,Y 495.764,Z 377.225,A -85,B 0,C 180,E1 -6169.301,E2 -6169.301} C_VEL
LIN {X 0,Y 495.73,Z 377.237,A -85,B 0,C 180,E1 -6172.44,E2 -6172.44} C_VEL
LIN {X 0,Y 495.785,Z 377.224,A -85,B 0,C 180,E1 -6175.458,E2 -6175.458} C_VEL
LIN {X 0,Y 495.758,Z 377.232,A -85,B 0,C 180,E1 -6178.365,E2 -6178.365} C_VEL
LIN {X 0,Y 495.788,Z 377.226,A -85,B 0,C 180,E1 -6181.508,E2 -6181.508} C_VEL
LIN {X 0,Y 495.8,Z 377.228,A -85,B 0,C 180,E1 -6183.933,E2 -6183.933} C_VEL
LIN {X 0,Y 495.836,Z 377.323,A -85,B 0,C 180,E1 -6185.786,E2 -6185.786} C_VEL
LIN {X 0,Y 497.414,Z 386.364,A -85,B 0,C 180,E1 -6187.575,E2 -6187.575} C_VEL
LIN {X 0,Y 497.219,Z 394.343,A -85,B 0,C 180,E1 -6189.013,E2 -6189.013} C_VEL
LIN {X 0,Y 496.642,Z 411.648,A -85,B 0,C 180,E1 -6192.075,E2 -6192.075} C_VEL
LIN {X 0,Y 496.323,Z 422.646,A -85,B 0,C 180,E1 -6193.948,E2 -6193.948} C_VEL
LIN {X 0,Y 498.532,Z 436.668,A -85,B 0,C 180,E1 -6194.254,E2 -6194.254} C_VEL
LIN {X 0,Y 498.034,Z 530.019,A -85,B 0,C 180,E1 -6195.625,E2 -6195.625} C_VEL
LIN {X 0,Y 497.718,Z 543.375,A -85,B 0,C 180,E1 -6195.981,E2 -6195.981} C_VEL
LIN {X 0,Y 497.403,Z 555.577,A -85,B 0,C 180,E1 -6196.467,E2 -6196.467} C_VEL
LIN {X 0,Y 497.035,Z 567.69,A -85,B 0,C 180,E1 -6197.12,E2 -6197.12} C_VEL
LIN {X 0,Y 496.657,Z 579.489,A -85,B 0,C 180,E1 -6197.953,E2 -6197.953} C_VEL
LIN {X 0,Y 496.276,Z 589.935,A -85,B 0,C 180,E1 -6198.875,E2 -6198.875} C_VEL
LIN {X 0,Y 495.927,Z 598.472,A -85,B 0,C 180,E1 -6199.797,E2 -6199.797} C_VEL
LIN {X 0,Y 495.65,Z 606.349,A -85,B 0,C 180,E1 -6200.821,E2 -6200.821} C_VEL
LIN {X 0,Y 495.383,Z 614.039,A -85,B 0,C 180,E1 -6202.05,E2 -6202.05} C_VEL
LIN {X 0,Y 495.164,Z 621.124,A -85,B 0,C 180,E1 -6203.481,E2 -6203.481} C_VEL
LIN {X 0,Y 495.116,Z 625.838,A -85,B 0,C 180,E1 -6204.706,E2 -6204.706} C_VEL
LIN {X 0,Y 495.034,Z 629.439,A -85,B 0,C 180,E1 -6205.93,E2 -6205.93} C_VEL
LIN {X 0,Y 495.042,Z 631.297,A -85,B 0,C 180,E1 -6206.745,E2 -6206.745} C_VEL
LIN {X 0,Y 494.961,Z 633.682,A -85,B 0,C 180,E1 -6208.373,E2 -6208.373} C_VEL
LIN {X 0,Y 494.898,Z 634.505,A -85,B 0,C 180,E1 -6210,E2 -6210} C_VEL
LIN {X 0,Y 494.961,Z 633.687,A -85,B 0,C 180,E1 -6211.627,E2 -6211.627} C_VEL
LIN {X 0,Y 495.042,Z 631.305,A -85,B 0,C 180,E1 -6213.256,E2 -6213.256} C_VEL
LIN {X 0,Y 495.01,Z 628.378,A -85,B 0,C 180,E1 -6214.479,E2 -6214.479} C_VEL
LIN {X 0,Y 495.152,Z 624.417,A -85,B 0,C 180,E1 -6215.702,E2 -6215.702} C_VEL
LIN {X 0,Y 495.257,Z 618.32,A -85,B 0,C 180,E1 -6217.133,E2 -6217.133} C_VEL
LIN {X 0,Y 495.459,Z 611.656,A -85,B 0,C 180,E1 -6218.36,E2 -6218.36} C_VEL
LIN {X 0,Y 495.739,Z 603.386,A -85,B 0,C 180,E1 -6219.589,E2 -6219.589} C_VEL
LIN {X 0,Y 496.044,Z 594.905,A -85,B 0,C 180,E1 -6220.614,E2 -6220.614} C_VEL
LIN {X 0,Y 496.466,Z 584.423,A -85,B 0,C 180,E1 -6221.638,E2 -6221.638} C_VEL
LIN {X 0,Y 496.84,Z 573.563,A -85,B 0,C 180,E1 -6222.493,E2 -6222.493} C_VEL
LIN {X 0,Y 497.177,Z 562.67,A -85,B 0,C 180,E1 -6223.176,E2 -6223.176} C_VEL
LIN {X 0,Y 497.568,Z 550.975,A -85,B 0,C 180,E1 -6223.737,E2 -6223.737} C_VEL
LIN {X 0,Y 497.844,Z 538.407,A -85,B 0,C 180,E1 -6224.172,E2 -6224.172} C_VEL
LIN {X 0,Y 498.076,Z 525.631,A -85,B 0,C 180,E1 -6224.452,E2 -6224.452} C_VEL
LIN {X 0,Y 498.487,Z 435.719,A -85,B 0,C 180,E1 -6225.761,E2 -6225.761} C_VEL
LIN {X 0,Y 496.313,Z 422.713,A -85,B 0,C 180,E1 -6226.044,E2 -6226.044} C_VEL
LIN {X 0,Y 496.583,Z 412.839,A -85,B 0,C 180,E1 -6227.715,E2 -6227.715} C_VEL
LIN {X 0,Y 497.118,Z 395.893,A -85,B 0,C 180,E1 -6230.697,E2 -6230.697} C_VEL
LIN {X 0,Y 497.394,Z 386.192,A -85,B 0,C 180,E1 -6232.426,E2 -6232.426} C_VEL
LIN {X 0,Y 495.827,Z 377.295,A -85,B 0,C 180,E1 -6234.159,E2 -6234.159} C_VEL
LIN {X 0,Y 495.815,Z 377.223,A -85,B 0,C 180,E1 -6236.974,E2 -6236.974} C_VEL
LIN {X 0,Y 495.766,Z 377.227,A -85,B 0,C 180,E1 -6240.147,E2 -6240.147} C_VEL
LIN {X 0,Y 495.794,Z 377.228,A -85,B 0,C 180,E1 -6243.244,E2 -6243.244} C_VEL
LIN {X 0,Y 495.729,Z 377.231,A -85,B 0,C 180,E1 -6246.09,E2 -6246.09} C_VEL
LIN {X 0,Y 495.764,Z 377.228,A -85,B 0,C 180,E1 -6248.768,E2 -6248.768} C_VEL
LIN {X 0,Y 495.776,Z 377.227,A -85,B 0,C 180,E1 -6251.778,E2 -6251.778} C_VEL
LIN {X 0,Y 495.747,Z 377.234,A -85,B 0,C 180,E1 -6255.139,E2 -6255.139} C_VEL
LIN {X 0,Y 495.783,Z 377.225,A -85,B 0,C 180,E1 -6258.221,E2 -6258.221} C_VEL
LIN {X 0,Y 495.776,Z 377.233,A -85,B 0,C 180,E1 -6261.229,E2 -6261.229} C_VEL
LIN {X 0,Y 495.754,Z 377.23,A -85,B 0,C 180,E1 -6264.463,E2 -6264.463} C_VEL
LIN {X 0,Y 495.765,Z 377.23,A -85,B 0,C 180,E1 -6267.405,E2 -6267.405} C_VEL
LIN {X 0,Y 495.762,Z 377.229,A -85,B 0,C 180,E1 -6270.253,E2 -6270.253} C_VEL
LIN {X 0,Y 495.829,Z 377.223,A -85,B 0,C 180,E1 -6273.248,E2 -6273.248} C_VEL
LIN {X 0,Y 495.747,Z 377.23,A -85,B 0,C 180,E1 -6275.725,E2 -6275.725} C_VEL
LIN {X 0,Y 495.738,Z 377.234,A -85,B 0,C 180,E1 -6278.371,E2 -6278.371} C_VEL
LIN {X 0,Y 495.78,Z 377.231,A -85,B 0,C 180,E1 -6280.971,E2 -6280.971} C_VEL
LIN {X 0,Y 495.775,Z 377.227,A -85,B 0,C 180,E1 -6283.53,E2 -6283.53} C_VEL
LIN {X 0,Y 495.788,Z 377.227,A -85,B 0,C 180,E1 -6286.055,E2 -6286.055} C_VEL
LIN {X 0,Y 495.845,Z 377.221,A -85,B 0,C 180,E1 -6288.555,E2 -6288.555} C_VEL
LIN {X 0,Y 495.867,Z 377.216,A -85,B 0,C 180,E1 -6291.852,E2 -6291.852} C_VEL
LIN {X 0,Y 495.89,Z 377.216,A -85,B 0,C 180,E1 -6294.306,E2 -6294.306} C_VEL
LIN {X 0,Y 495.987,Z 377.201,A -85,B 0,C 180,E1 -6297.564,E2 -6297.564} C_VEL
LIN {X 0,Y 495.991,Z 377.204,A -85,B 0,C 180,E1 -6300,E2 -6300} C_VEL
LIN {X 0,Y 495.987,Z 377.204,A -85,B 0,C 180,E1 -6302.436,E2 -6302.436} C_VEL
LIN {X 0,Y 495.89,Z 377.214,A -85,B 0,C 180,E1 -6305.693,E2 -6305.693} C_VEL
LIN {X 0,Y 495.866,Z 377.219,A -85,B 0,C 180,E1 -6308.148,E2 -6308.148} C_VEL
LIN {X 0,Y 495.845,Z 377.219,A -85,B 0,C 180,E1 -6311.445,E2 -6311.445} C_VEL
LIN {X 0,Y 495.784,Z 377.227,A -85,B 0,C 180,E1 -6314.783,E2 -6314.783} C_VEL
LIN {X 0,Y 495.783,Z 377.227,A -85,B 0,C 180,E1 -6317.319,E2 -6317.319} C_VEL
LIN {X 0,Y 495.773,Z 377.231,A -85,B 0,C 180,E1 -6319.89,E2 -6319.89} C_VEL
LIN {X 0,Y 495.76,Z 377.229,A -85,B 0,C 180,E1 -6322.863,E2 -6322.863} C_VEL
LIN {X 0,Y 495.794,Z 377.227,A -85,B 0,C 180,E1 -6326.068,E2 -6326.068} C_VEL
LIN {X 0,Y 495.775,Z 377.227,A -85,B 0,C 180,E1 -6328.815,E2 -6328.815} C_VEL
LIN {X 0,Y 495.755,Z 377.233,A -85,B 0,C 180,E1 -6331.727,E2 -6331.727} C_VEL
LIN {X 0,Y 495.773,Z 377.227,A -85,B 0,C 180,E1 -6334.696,E2 -6334.696} C_VEL
LIN {X 0,Y 495.728,Z 377.238,A -85,B 0,C 180,E1 -6337.562,E2 -6337.562} C_VEL
LIN {X 0,Y 495.763,Z 377.228,A -85,B 0,C 180,E1 -6340.7,E2 -6340.7} C_VEL
LIN {X 0,Y 495.732,Z 377.235,A -85,B 0,C 180,E1 -6343.696,E2 -6343.696} C_VEL
LIN {X 0,Y 495.726,Z 377.233,A -85,B 0,C 180,E1 -6346.306,E2 -6346.306} C_VEL
LIN {X 0,Y 495.778,Z 377.232,A -85,B 0,C 180,E1 -6349.302,E2 -6349.302} C_VEL
LIN {X 0,Y 495.73,Z 377.232,A -85,B 0,C 180,E1 -6352.439,E2 -6352.439} C_VEL
LIN {X 0,Y 495.785,Z 377.229,A -85,B 0,C 180,E1 -6355.458,E2 -6355.458} C_VEL
LIN {X 0,Y 495.756,Z 377.228,A -85,B 0,C 180,E1 -6358.364,E2 -6358.364} C_VEL
LIN {X 0,Y 495.753,Z 377.23,A -85,B 0,C 180,E1 -6360.767,E2 -6360.767} C_VEL
LIN {X 0,Y 495.097,Z 377.317,A -85,B 0,C 180,E1 -6361.446,E2 -6361.446} C_VEL
LIN {X 0,Y 492.24,Z 377.67,A -85,B 0,C 180,E1 -6362.549,E2 -6362.549} C_VEL
LIN {X 0,Y 489.831,Z 377.97,A -85,B 0,C 180,E1 -6363.437,E2 -6363.437} C_VEL
LIN {X 0,Y 488.815,Z 378.093,A -85,B 0,C 180,E1 -6364.124,E2 -6364.124} C_VEL
LIN {X 0,Y 488.743,Z 378.101,A -85,B 0,C 180,E1 -6364.356,E2 -6364.356} C_VEL
LIN {X 0,Y 488.724,Z 378.111,A -85,B 0,C 180,E1 -6367.153,E2 -6367.153} C_VEL
LIN {X 0,Y 488.726,Z 378.104,A -85,B 0,C 180,E1 -6369.811,E2 -6369.811} C_VEL
LIN {X 0,Y 488.731,Z 378.104,A -85,B 0,C 180,E1 -6372.423,E2 -6372.423} C_VEL
LIN {X 0,Y 488.764,Z 378.106,A -85,B 0,C 180,E1 -6375,E2 -6375} C_VEL
LIN {X 0,Y 488.808,Z 378.098,A -85,B 0,C 180,E1 -6378.388,E2 -6378.388} C_VEL
LIN {X 0,Y 488.791,Z 378.207,A -85,B 0,C 180,E1 -6380.535,E2 -6380.535} C_VEL
LIN {X 0,Y 490.066,Z 385.385,A -85,B 0,C 180,E1 -6382.062,E2 -6382.062} C_VEL
LIN {X 0,Y 489.745,Z 395.411,A -85,B 0,C 180,E1 -6384.028,E2 -6384.028} C_VEL
LIN {X 0,Y 489.328,Z 409.659,A -85,B 0,C 180,E1 -6386.758,E2 -6386.758} C_VEL
LIN {X 0,Y 490.019,Z 413.587,A -85,B 0,C 180,E1 -6386.882,E2 -6386.882} C_VEL
LIN {X 0,Y 491.786,Z 423.157,A -85,B 0,C 180,E1 -6387.082,E2 -6387.082} C_VEL
LIN {X 0,Y 491.116,Z 517.448,A -85,B 0,C 180,E1 -6388.488,E2 -6388.488} C_VEL
LIN {X 0,Y 490.862,Z 531.064,A -85,B 0,C 180,E1 -6388.872,E2 -6388.872} C_VEL
LIN {X 0,Y 490.54,Z 543.336,A -85,B 0,C 180,E1 -6389.384,E2 -6389.384} C_VEL
LIN {X 0,Y 490.088,Z 555.912,A -85,B 0,C 180,E1 -6390.102,E2 -6390.102} C_VEL
LIN {X 0,Y 489.629,Z 567.097,A -85,B 0,C 180,E1 -6390.925,E2 -6390.925} C_VEL
LIN {X 0,Y 489.274,Z 577.183,A -85,B 0,C 180,E1 -6391.852,E2 -6391.852} C_VEL
LIN {X 0,Y 488.851,Z 586.299,A -85,B 0,C 180,E1 -6392.884,E2 -6392.884} C_VEL
LIN {X 0,Y 488.559,Z 595.17,A -85,B 0,C 180,E1 -6394.124,E2 -6394.124} C_VEL
LIN {X 0,Y 488.218,Z 602.359,A -85,B 0,C 180,E1 -6395.369,E2 -6395.369} C_VEL
LIN {X 0,Y 488.181,Z 608.085,A -85,B 0,C 180,E1 -6396.613,E2 -6396.613} C_VEL
LIN {X 0,Y 488.014,Z 612.626,A -85,B 0,C 180,E1 -6397.863,E2 -6397.863} C_VEL
LIN {X 0,Y 487.901,Z 616.085,A -85,B 0,C 180,E1 -6399.117,E2 -6399.117} C_VEL
LIN {X 0,Y 487.849,Z 617.806,A -85,B 0,C 180,E1 -6399.954,E2 -6399.954} C_VEL
LIN {X 0,Y 487.911,Z 620.018,A -85,B 0,C 180,E1 -6401.624,E2 -6401.624} C_VEL
LIN {X 0,Y 487.834,Z 620.511,A -85,B 0,C 180,E1 -6402.479,E2 -6402.479} C_VEL
LIN {X 0,Y 487.8,Z 620.567,A -85,B 0,C 180,E1 -6403.327,E2 -6403.327} C_VEL
LIN {X 0,Y 487.833,Z 620.224,A -85,B 0,C 180,E1 -6404.176,E2 -6404.176} C_VEL
LIN {X 0,Y 487.86,Z 619.3,A -85,B 0,C 180,E1 -6405.163,E2 -6405.163} C_VEL
LIN {X 0,Y 487.864,Z 616.586,A -85,B 0,C 180,E1 -6406.744,E2 -6406.744} C_VEL
LIN {X 0,Y 487.986,Z 613.03,A -85,B 0,C 180,E1 -6408.096,E2 -6408.096} C_VEL
LIN {X 0,Y 488.108,Z 608.642,A -85,B 0,C 180,E1 -6409.339,E2 -6409.339} C_VEL
LIN {X 0,Y 488.319,Z 602.521,A -85,B 0,C 180,E1 -6410.691,E2 -6410.691} C_VEL
LIN {X 0,Y 488.554,Z 595.207,A -85,B 0,C 180,E1 -6411.963,E2 -6411.963} C_VEL
LIN {X 0,Y 488.911,Z 586.782,A -85,B 0,C 180,E1 -6413.146,E2 -6413.146} C_VEL
LIN {X 0,Y 489.293,Z 576.833,A -85,B 0,C 180,E1 -6414.277,E2 -6414.277} C_VEL
LIN {X 0,Y 489.666,Z 566.762,A -85,B 0,C 180,E1 -6415.195,E2 -6415.195} C_VEL
LIN {X 0,Y 490.12,Z 555.048,A -85,B 0,C 180,E1 -6416.048,E2 -6416.048} C_VEL
LIN {X 0,Y 490.547,Z 543.321,A -85,B 0,C 180,E1 -6416.711,E2 -6416.711} C_VEL
LIN {X 0,Y 490.909,Z 530.228,A -85,B 0,C 180,E1 -6417.251,E2 -6417.251} C_VEL
LIN {X 0,Y 491.143,Z 517.088,A -85,B 0,C 180,E1 -6417.614,E2 -6417.614} C_VEL
LIN {X 0,Y 491.755,Z 423.123,A -85,B 0,C 180,E1 -6419.027,E2 -6419.027} C_VEL
LIN {X 0,Y 489.429,Z 410.058,A -85,B 0,C 180,E1 -6419.321,E2 -6419.321} C_VEL
LIN {X 0,Y 489.379,Z 408.964,A -85,B 0,C 180,E1 -6419.462,E2 -6419.462} C_VEL
LIN {X 0,Y 490.01,Z 391.945,A -85,B 0,C 180,E1 -6422.784,E2 -6422.784} C_VEL
LIN {X 0,Y 490.17,Z 385.848,A -85,B 0,C 180,E1 -6423.998,E2 -6423.998} C_VEL
LIN {X 0,Y 488.72,Z 378.14,A -85,B 0,C 180,E1 -6425.698,E2 -6425.698} C_VEL
LIN {X 0,Y 488.745,Z 378.107,A -85,B 0,C 180,E1 -6429.249,E2 -6429.249} C_VEL
LIN {X 0,Y 488.731,Z 378.106,A -85,B 0,C 180,E1 -6432.52,E2 -6432.52} C_VEL
LIN {X 0,Y 488.697,Z 378.108,A -85,B 0,C 180,E1 -6435.975,E2 -6435.975} C_VEL
LIN {X 0,Y 488.722,Z 378.103,A -85,B 0,C 180,E1 -6438.586,E2 -6438.586} C_VEL
LIN {X 0,Y 488.741,Z 378.104,A -85,B 0,C 180,E1 -6440.94,E2 -6440.94} C_VEL
LIN {X 0,Y 488.68,Z 378.109,A -85,B 0,C 180,E1 -6443.868,E2 -6443.868} C_VEL
LIN {X 0,Y 488.732,Z 378.105,A -85,B 0,C 180,E1 -6446.877,E2 -6446.877} C_VEL
LIN {X 0,Y 488.727,Z 378.096,A -85,B 0,C 180,E1 -6449.781,E2 -6449.781} C_VEL
LIN {X 0,Y 488.791,Z 378.103,A -85,B 0,C 180,E1 -6453.054,E2 -6453.054} C_VEL
LIN {X 0,Y 488.692,Z 378.108,A -85,B 0,C 180,E1 -6456.255,E2 -6456.255} C_VEL
LIN {X 0,Y 488.738,Z 378.107,A -85,B 0,C 180,E1 -6459.175,E2 -6459.175} C_VEL
LIN {X 0,Y 488.75,Z 378.098,A -85,B 0,C 180,E1 -6461.627,E2 -6461.627} C_VEL
LIN {X 0,Y 488.752,Z 378.103,A -85,B 0,C 180,E1 -6464.999,E2 -6464.999} C_VEL
LIN {X 0,Y 488.824,Z 378.093,A -85,B 0,C 180,E1 -6468.388,E2 -6468.388} C_VEL
LIN {X 0,Y 488.809,Z 378.093,A -85,B 0,C 180,E1 -6471.734,E2 -6471.734} C_VEL
LIN {X 0,Y 488.853,Z 378.085,A -85,B 0,C 180,E1 -6474.224,E2 -6474.224} C_VEL
LIN {X 0,Y 488.958,Z 378.074,A -85,B 0,C 180,E1 -6477.529,E2 -6477.529} C_VEL
LIN {X 0,Y 488.959,Z 378.072,A -85,B 0,C 180,E1 -6480,E2 -6480} C_VEL
LIN {X 0,Y 488.953,Z 378.078,A -85,B 0,C 180,E1 -6482.471,E2 -6482.471} C_VEL
LIN {X 0,Y 488.853,Z 378.087,A -85,B 0,C 180,E1 -6485.776,E2 -6485.776} C_VEL
LIN {X 0,Y 488.809,Z 378.093,A -85,B 0,C 180,E1 -6488.267,E2 -6488.267} C_VEL
LIN {X 0,Y 488.821,Z 378.091,A -85,B 0,C 180,E1 -6491.612,E2 -6491.612} C_VEL
LIN {X 0,Y 488.753,Z 378.104,A -85,B 0,C 180,E1 -6495.001,E2 -6495.001} C_VEL
LIN {X 0,Y 488.746,Z 378.103,A -85,B 0,C 180,E1 -6498.443,E2 -6498.443} C_VEL
LIN {X 0,Y 488.704,Z 378.108,A -85,B 0,C 180,E1 -6501.071,E2 -6501.071} C_VEL
LIN {X 0,Y 488.693,Z 378.106,A -85,B 0,C 180,E1 -6503.746,E2 -6503.746} C_VEL
LIN {X 0,Y 488.791,Z 378.098,A -85,B 0,C 180,E1 -6506.946,E2 -6506.946} C_VEL
LIN {X 0,Y 488.703,Z 378.11,A -85,B 0,C 180,E1 -6510.364,E2 -6510.364} C_VEL
LIN {X 0,Y 488.729,Z 378.101,A -85,B 0,C 180,E1 -6513.485,E2 -6513.485} C_VEL
LIN {X 0,Y 488.684,Z 378.114,A -85,B 0,C 180,E1 -6516.357,E2 -6516.357} C_VEL
LIN {X 0,Y 488.737,Z 378.102,A -85,B 0,C 180,E1 -6519.251,E2 -6519.251} C_VEL
LIN {X 0,Y 488.731,Z 378.102,A -85,B 0,C 180,E1 -6522.522,E2 -6522.522} C_VEL
LIN {X 0,Y 488.708,Z 378.104,A -85,B 0,C 180,E1 -6525.2,E2 -6525.2} C_VEL
LIN {X 0,Y 488.72,Z 378.11,A -85,B 0,C 180,E1 -6528.399,E2 -6528.399} C_VEL
LIN {X 0,Y 488.702,Z 378.11,A -85,B 0,C 180,E1 -6530.948,E2 -6530.948} C_VEL
LIN {X 0,Y 488.684,Z 378.107,A -85,B 0,C 180,E1 -6533.87,E2 -6533.87} C_VEL
LIN {X 0,Y 488.738,Z 378.106,A -85,B 0,C 180,E1 -6536.878,E2 -6536.878} C_VEL
LIN {X 0,Y 488.723,Z 378.107,A -85,B 0,C 180,E1 -6539.782,E2 -6539.782} C_VEL
LIN {X 0,Y 488.799,Z 378.098,A -85,B 0,C 180,E1 -6543.055,E2 -6543.055} C_VEL
LIN {X 0,Y 488.787,Z 378.225,A -85,B 0,C 180,E1 -6545.583,E2 -6545.583} C_VEL
LIN {X 0,Y 490.46,Z 387.571,A -85,B 0,C 180,E1 -6547.462,E2 -6547.462} C_VEL
LIN {X 0,Y 490.372,Z 393.107,A -85,B 0,C 180,E1 -6548.481,E2 -6548.481} C_VEL
LIN {X 0,Y 489.692,Z 411.595,A -85,B 0,C 180,E1 -6551.812,E2 -6551.812} C_VEL
LIN {X 0,Y 489.349,Z 422.401,A -85,B 0,C 180,E1 -6553.694,E2 -6553.694} C_VEL
LIN {X 0,Y 491.434,Z 435.082,A -85,B 0,C 180,E1 -6553.988,E2 -6553.988} C_VEL
LIN {X 0,Y 491.751,Z 442.812,A -85,B 0,C 180,E1 -6554.116,E2 -6554.116} C_VEL
LIN {X 0,Y 491.174,Z 529.965,A -85,B 0,C 180,E1 -6555.42,E2 -6555.42} C_VEL
LIN {X 0,Y 490.818,Z 543.296,A -85,B 0,C 180,E1 -6555.78,E2 -6555.78} C_VEL
LIN {X 0,Y 490.465,Z 556.612,A -85,B 0,C 180,E1 -6556.324,E2 -6556.324} C_VEL
LIN {X 0,Y 490.11,Z 567.586,A -85,B 0,C 180,E1 -6556.935,E2 -6556.935} C_VEL
LIN {X 0,Y 489.69,Z 579.383,A -85,B 0,C 180,E1 -6557.779,E2 -6557.779} C_VEL
LIN {X 0,Y 489.292,Z 589.825,A -85,B 0,C 180,E1 -6558.715,E2 -6558.715} C_VEL
LIN {X 0,Y 488.89,Z 598.362,A -85,B 0,C 180,E1 -6559.649,E2 -6559.649} C_VEL
LIN {X 0,Y 488.618,Z 606.24,A -85,B 0,C 180,E1 -6560.688,E2 -6560.688} C_VEL
LIN {X 0,Y 488.329,Z 613.932,A -85,B 0,C 180,E1 -6561.934,E2 -6561.934} C_VEL
LIN {X 0,Y 488.1,Z 621.02,A -85,B 0,C 180,E1 -6563.386,E2 -6563.386} C_VEL
LIN {X 0,Y 488.05,Z 625.735,A -85,B 0,C 180,E1 -6564.63,E2 -6564.63} C_VEL
LIN {X 0,Y 487.929,Z 629.336,A -85,B 0,C 180,E1 -6565.87,E2 -6565.87} C_VEL
LIN {X 0,Y 487.964,Z 631.195,A -85,B 0,C 180,E1 -6566.698,E2 -6566.698} C_VEL
LIN {X 0,Y 487.889,Z 633.582,A -85,B 0,C 180,E1 -6568.349,E2 -6568.349} C_VEL
LIN {X 0,Y 487.819,Z 634.405,A -85,B 0,C 180,E1 -6570,E2 -6570} C_VEL
LIN {X 0,Y 487.889,Z 633.587,A -85,B 0,C 180,E1 -6571.651,E2 -6571.651} C_VEL
LIN {X 0,Y 487.965,Z 631.205,A -85,B 0,C 180,E1 -6573.303,E2 -6573.303} C_VEL
LIN {X 0,Y 487.922,Z 628.277,A -85,B 0,C 180,E1 -6574.544,E2 -6574.544} C_VEL
LIN {X 0,Y 488.069,Z 624.315,A -85,B 0,C 180,E1 -6575.785,E2 -6575.785} C_VEL
LIN {X 0,Y 488.184,Z 618.217,A -85,B 0,C 180,E1 -6577.237,E2 -6577.237} C_VEL
LIN {X 0,Y 488.424,Z 611.552,A -85,B 0,C 180,E1 -6578.481,E2 -6578.481} C_VEL
LIN {X 0,Y 488.722,Z 603.281,A -85,B 0,C 180,E1 -6579.728,E2 -6579.728} C_VEL
LIN {X 0,Y 489.038,Z 594.798,A -85,B 0,C 180,E1 -6580.767,E2 -6580.767} C_VEL
LIN {X 0,Y 489.51,Z 584.314,A -85,B 0,C 180,E1 -6581.805,E2 -6581.805} C_VEL
LIN {X 0,Y 489.904,Z 572.99,A -85,B 0,C 180,E1 -6582.706,E2 -6582.706} C_VEL
LIN {X 0,Y 490.31,Z 560.608,A -85,B 0,C 180,E1 -6583.469,E2 -6583.469} C_VEL
LIN {X 0,Y 490.727,Z 548.228,A -85,B 0,C 180,E1 -6584.038,E2 -6584.038} C_VEL
LIN {X 0,Y 491.065,Z 535.488,A -85,B 0,C 180,E1 -6584.451,E2 -6584.451} C_VEL
LIN {X 0,Y 491.202,Z 522.048,A -85,B 0,C 180,E1 -6584.712,E2 -6584.712} C_VEL
LIN {X 0,Y 491.65,Z 436.425,A -85,B 0,C 180,E1 -6585.971,E2 -6585.971} C_VEL
LIN {X 0,Y 489.322,Z 422.5,A -85,B 0,C 180,E1 -6586.278,E2 -6586.278} C_VEL
LIN {X 0,Y 489.86,Z 405.442,A -85,B 0,C 180,E1 -6589.267,E2 -6589.267} C_VEL
LIN {X 0,Y 490.495,Z 388.464,A -85,B 0,C 180,E1 -6592.315,E2 -6592.315} C_VEL
LIN {X 0,Y 488.802,Z 378.229,A -85,B 0,C 180,E1 -6594.303,E2 -6594.303} C_VEL
LIN {X 0,Y 488.748,Z 378.108,A -85,B 0,C 180,E1 -6597.396,E2 -6597.396} C_VEL
LIN {X 0,Y 488.711,Z 378.105,A -85,B 0,C 180,E1 -6600.363,E2 -6600.363} C_VEL
LIN {X 0,Y 488.736,Z 378.109,A -85,B 0,C 180,E1 -6603.484,E2 -6603.484} C_VEL
LIN {X 0,Y 488.69,Z 378.108,A -85,B 0,C 180,E1 -6606.355,E2 -6606.355} C_VEL
LIN {X 0,Y 488.701,Z 378.112,A -85,B 0,C 180,E1 -6609.254,E2 -6609.254} C_VEL
LIN {X 0,Y 488.723,Z 378.108,A -85,B 0,C 180,E1 -6611.601,E2 -6611.601} C_VEL
LIN {X 0,Y 488.71,Z 378.108,A -85,B 0,C 180,E1 -6614.801,E2 -6614.801} C_VEL
LIN {X 0,Y 488.732,Z 378.107,A -85,B 0,C 180,E1 -6617.479,E2 -6617.479} C_VEL
LIN {X 0,Y 488.746,Z 378.104,A -85,B 0,C 180,E1 -6620.75,E2 -6620.75} C_VEL
LIN {X 0,Y 488.682,Z 378.11,A -85,B 0,C 180,E1 -6623.868,E2 -6623.868} C_VEL
LIN {X 0,Y 488.735,Z 378.107,A -85,B 0,C 180,E1 -6626.877,E2 -6626.877} C_VEL
LIN {X 0,Y 488.72,Z 378.106,A -85,B 0,C 180,E1 -6629.78,E2 -6629.78} C_VEL
LIN {X 0,Y 488.794,Z 378.102,A -85,B 0,C 180,E1 -6633.054,E2 -6633.054} C_VEL
LIN {X 0,Y 488.688,Z 378.111,A -85,B 0,C 180,E1 -6636.254,E2 -6636.254} C_VEL
LIN {X 0,Y 488.74,Z 378.106,A -85,B 0,C 180,E1 -6639.175,E2 -6639.175} C_VEL
LIN {X 0,Y 488.754,Z 378.102,A -85,B 0,C 180,E1 -6641.627,E2 -6641.627} C_VEL
LIN {X 0,Y 488.756,Z 378.105,A -85,B 0,C 180,E1 -6644.999,E2 -6644.999} C_VEL
LIN {X 0,Y 488.799,Z 378.099,A -85,B 0,C 180,E1 -6648.387,E2 -6648.387} C_VEL
LIN {X 0,Y 488.811,Z 378.095,A -85,B 0,C 180,E1 -6651.733,E2 -6651.733} C_VEL
LIN {X 0,Y 488.849,Z 378.093,A -85,B 0,C 180,E1 -6654.224,E2 -6654.224} C_VEL
LIN {X 0,Y 488.955,Z 378.077,A -85,B 0,C 180,E1 -6657.529,E2 -6657.529} C_VEL
LIN {X 0,Y 488.949,Z 378.08,A -85,B 0,C 180,E1 -6660.824,E2 -6660.824} C_VEL
LIN {X 0,Y 488.955,Z 378.08,A -85,B 0,C 180,E1 -6662.471,E2 -6662.471} C_VEL
LIN {X 0,Y 488.849,Z 378.092,A -85,B 0,C 180,E1 -6665.776,E2 -6665.776} C_VEL
LIN {X 0,Y 488.811,Z 378.097,A -85,B 0,C 180,E1 -6668.266,E2 -6668.266} C_VEL
LIN {X 0,Y 488.799,Z 378.098,A -85,B 0,C 180,E1 -6671.613,E2 -6671.613} C_VEL
LIN {X 0,Y 488.756,Z 378.102,A -85,B 0,C 180,E1 -6675.001,E2 -6675.001} C_VEL
LIN {X 0,Y 488.749,Z 378.105,A -85,B 0,C 180,E1 -6678.442,E2 -6678.442} C_VEL
LIN {X 0,Y 488.701,Z 378.108,A -85,B 0,C 180,E1 -6681.071,E2 -6681.071} C_VEL
LIN {X 0,Y 488.689,Z 378.114,A -85,B 0,C 180,E1 -6683.746,E2 -6683.746} C_VEL
LIN {X 0,Y 488.794,Z 378.097,A -85,B 0,C 180,E1 -6686.946,E2 -6686.946} C_VEL
LIN {X 0,Y 488.714,Z 378.109,A -85,B 0,C 180,E1 -6690.365,E2 -6690.365} C_VEL
LIN {X 0,Y 488.732,Z 378.109,A -85,B 0,C 180,E1 -6693.485,E2 -6693.485} C_VEL
LIN {X 0,Y 488.685,Z 378.111,A -85,B 0,C 180,E1 -6696.356,E2 -6696.356} C_VEL
LIN {X 0,Y 488.698,Z 378.111,A -85,B 0,C 180,E1 -6699.255,E2 -6699.255} C_VEL
LIN {X 0,Y 488.72,Z 378.11,A -85,B 0,C 180,E1 -6701.602,E2 -6701.602} C_VEL
LIN {X 0,Y 488.709,Z 378.107,A -85,B 0,C 180,E1 -6704.802,E2 -6704.802} C_VEL
LIN {X 0,Y 488.689,Z 378.114,A -85,B 0,C 180,E1 -6707.475,E2 -6707.475} C_VEL
LIN {X 0,Y 488.731,Z 378.107,A -85,B 0,C 180,E1 -6709.677,E2 -6709.677} C_VEL
LIN {X 0,Y 488.679,Z 378.11,A -85,B 0,C 180,E1 -6712.278,E2 -6712.278} C_VEL
LIN {X 0,Y 488.728,Z 378.108,A -85,B 0,C 180,E1 -6715.052,E2 -6715.052} C_VEL
LIN {X 0,Y 488.703,Z 378.108,A -85,B 0,C 180,E1 -6718.046,E2 -6718.046} C_VEL
LIN {X 0,Y 488.723,Z 378.106,A -85,B 0,C 180,E1 -6720.765,E2 -6720.765} C_VEL
LIN {X 0,Y 488.757,Z 378.103,A -85,B 0,C 180,E1 -6723.528,E2 -6723.528} C_VEL
LIN {X 0,Y 488.743,Z 378.101,A -85,B 0,C 180,E1 -6724.356,E2 -6724.356} C_VEL
LIN {X 0,Y 488.099,Z 378.188,A -85,B 0,C 180,E1 -6725.044,E2 -6725.044} C_VEL
LIN {X 0,Y 485.23,Z 378.543,A -85,B 0,C 180,E1 -6726.16,E2 -6726.16} C_VEL
LIN {X 0,Y 482.782,Z 378.851,A -85,B 0,C 180,E1 -6727.06,E2 -6727.06} C_VEL
LIN {X 0,Y 481.724,Z 378.977,A -85,B 0,C 180,E1 -6727.755,E2 -6727.755} C_VEL
LIN {X 0,Y 481.636,Z 378.987,A -85,B 0,C 180,E1 -6727.991,E2 -6727.991} C_VEL
LIN {X 0,Y 481.706,Z 378.978,A -85,B 0,C 180,E1 -6730.393,E2 -6730.393} C_VEL
LIN {X 0,Y 481.69,Z 378.987,A -85,B 0,C 180,E1 -6733.034,E2 -6733.034} C_VEL
LIN {X 0,Y 481.691,Z 378.982,A -85,B 0,C 180,E1 -6735.639,E2 -6735.639} C_VEL
LIN {X 0,Y 481.753,Z 378.976,A -85,B 0,C 180,E1 -6738.215,E2 -6738.215} C_VEL
LIN {X 0,Y 481.744,Z 379.126,A -85,B 0,C 180,E1 -6740.395,E2 -6740.395} C_VEL
LIN {X 0,Y 483.076,Z 386.515,A -85,B 0,C 180,E1 -6741.972,E2 -6741.972} C_VEL
LIN {X 0,Y 482.741,Z 396.425,A -85,B 0,C 180,E1 -6743.941,E2 -6743.941} C_VEL
LIN {X 0,Y 482.349,Z 409.795,A -85,B 0,C 180,E1 -6746.528,E2 -6746.528} C_VEL
LIN {X 0,Y 483.317,Z 415.148,A -85,B 0,C 180,E1 -6746.68,E2 -6746.68} C_VEL
LIN {X 0,Y 484.877,Z 423.489,A -85,B 0,C 180,E1 -6746.858,E2 -6746.858} C_VEL
LIN {X 0,Y 484.252,Z 517.598,A -85,B 0,C 180,E1 -6748.285,E2 -6748.285} C_VEL
LIN {X 0,Y 483.977,Z 531.212,A -85,B 0,C 180,E1 -6748.674,E2 -6748.674} C_VEL
LIN {X 0,Y 483.606,Z 543.994,A -85,B 0,C 180,E1 -6749.219,E2 -6749.219} C_VEL
LIN {X 0,Y 483.188,Z 555.658,A -85,B 0,C 180,E1 -6749.896,E2 -6749.896} C_VEL
LIN {X 0,Y 482.68,Z 566.923,A -85,B 0,C 180,E1 -6750.73,E2 -6750.73} C_VEL
LIN {X 0,Y 482.299,Z 577.073,A -85,B 0,C 180,E1 -6751.67,E2 -6751.67} C_VEL
LIN {X 0,Y 481.84,Z 586.239,A -85,B 0,C 180,E1 -6752.717,E2 -6752.717} C_VEL
LIN {X 0,Y 481.503,Z 595.143,A -85,B 0,C 180,E1 -6753.975,E2 -6753.975} C_VEL
LIN {X 0,Y 481.149,Z 602.355,A -85,B 0,C 180,E1 -6755.238,E2 -6755.238} C_VEL
LIN {X 0,Y 481.089,Z 608.481,A -85,B 0,C 180,E1 -6756.596,E2 -6756.596} C_VEL
LIN {X 0,Y 480.91,Z 613.293,A -85,B 0,C 180,E1 -6757.98,E2 -6757.98} C_VEL
LIN {X 0,Y 480.789,Z 616.598,A -85,B 0,C 180,E1 -6759.253,E2 -6759.253} C_VEL
LIN {X 0,Y 480.755,Z 618.24,A -85,B 0,C 180,E1 -6760.103,E2 -6760.103} C_VEL
LIN {X 0,Y 480.808,Z 620.176,A -85,B 0,C 180,E1 -6761.666,E2 -6761.666} C_VEL
LIN {X 0,Y 480.746,Z 620.649,A -85,B 0,C 180,E1 -6762.667,E2 -6762.667} C_VEL
LIN {X 0,Y 480.701,Z 620.63,A -85,B 0,C 180,E1 -6763.528,E2 -6763.528} C_VEL
LIN {X 0,Y 480.729,Z 620.207,A -85,B 0,C 180,E1 -6764.39,E2 -6764.39} C_VEL
LIN {X 0,Y 480.752,Z 619.319,A -85,B 0,C 180,E1 -6765.256,E2 -6765.256} C_VEL
LIN {X 0,Y 480.727,Z 618.006,A -85,B 0,C 180,E1 -6766.127,E2 -6766.127} C_VEL
LIN {X 0,Y 480.848,Z 615.187,A -85,B 0,C 180,E1 -6767.434,E2 -6767.434} C_VEL
LIN {X 0,Y 480.965,Z 611.248,A -85,B 0,C 180,E1 -6768.751,E2 -6768.751} C_VEL
LIN {X 0,Y 481.122,Z 606.059,A -85,B 0,C 180,E1 -6770.076,E2 -6770.076} C_VEL
LIN {X 0,Y 481.383,Z 599.426,A -85,B 0,C 180,E1 -6771.406,E2 -6771.406} C_VEL
LIN {X 0,Y 481.706,Z 590.978,A -85,B 0,C 180,E1 -6772.744,E2 -6772.744} C_VEL
LIN {X 0,Y 482.141,Z 581.402,A -85,B 0,C 180,E1 -6773.962,E2 -6773.962} C_VEL
LIN {X 0,Y 482.541,Z 571.357,A -85,B 0,C 180,E1 -6774.984,E2 -6774.984} C_VEL
LIN {X 0,Y 483.039,Z 560.402,A -85,B 0,C 180,E1 -6775.879,E2 -6775.879} C_VEL
LIN {X 0,Y 483.362,Z 550.066,A -85,B 0,C 180,E1 -6776.557,E2 -6776.557} C_VEL
LIN {X 0,Y 483.838,Z 537.922,A -85,B 0,C 180,E1 -6777.17,E2 -6777.17} C_VEL
LIN {X 0,Y 484.152,Z 524.486,A -85,B 0,C 180,E1 -6777.649,E2 -6777.649} C_VEL
LIN {X 0,Y 484.389,Z 511.222,A -85,B 0,C 180,E1 -6777.941,E2 -6777.941} C_VEL
LIN {X 0,Y 484.977,Z 424.042,A -85,B 0,C 180,E1 -6779.253,E2 -6779.253} C_VEL
LIN {X 0,Y 482.429,Z 409.896,A -85,B 0,C 180,E1 -6779.59,E2 -6779.59} C_VEL
LIN {X 0,Y 482.991,Z 394.641,A -85,B 0,C 180,E1 -6782.573,E2 -6782.573} C_VEL
LIN {X 0,Y 483.233,Z 387.546,A -85,B 0,C 180,E1 -6784.005,E2 -6784.005} C_VEL
LIN {X 0,Y 481.667,Z 379.033,A -85,B 0,C 180,E1 -6785.899,E2 -6785.899} C_VEL
LIN {X 0,Y 481.716,Z 378.982,A -85,B 0,C 180,E1 -6789.354,E2 -6789.354} C_VEL
LIN {X 0,Y 481.67,Z 378.984,A -85,B 0,C 180,E1 -6792.157,E2 -6792.157} C_VEL
LIN {X 0,Y 481.655,Z 378.987,A -85,B 0,C 180,E1 -6794.456,E2 -6794.456} C_VEL
LIN {X 0,Y 481.684,Z 378.986,A -85,B 0,C 180,E1 -6796.845,E2 -6796.845} C_VEL
LIN {X 0,Y 481.687,Z 378.98,A -85,B 0,C 180,E1 -6800.061,E2 -6800.061} C_VEL
LIN {X 0,Y 481.625,Z 378.993,A -85,B 0,C 180,E1 -6803.253,E2 -6803.253} C_VEL
LIN {X 0,Y 481.702,Z 378.976,A -85,B 0,C 180,E1 -6806.329,E2 -6806.329} C_VEL
LIN {X 0,Y 481.657,Z 378.979,A -85,B 0,C 180,E1 -6809.414,E2 -6809.414} C_VEL
LIN {X 0,Y 481.695,Z 378.978,A -85,B 0,C 180,E1 -6812.168,E2 -6812.168} C_VEL
LIN {X 0,Y 481.711,Z 378.982,A -85,B 0,C 180,E1 -6814.97,E2 -6814.97} C_VEL
LIN {X 0,Y 481.651,Z 378.982,A -85,B 0,C 180,E1 -6817.705,E2 -6817.705} C_VEL
LIN {X 0,Y 481.7,Z 378.98,A -85,B 0,C 180,E1 -6820.393,E2 -6820.393} C_VEL
LIN {X 0,Y 481.683,Z 378.988,A -85,B 0,C 180,E1 -6823.034,E2 -6823.034} C_VEL
LIN {X 0,Y 481.682,Z 378.978,A -85,B 0,C 180,E1 -6825.639,E2 -6825.639} C_VEL
LIN {X 0,Y 481.786,Z 378.968,A -85,B 0,C 180,E1 -6828.216,E2 -6828.216} C_VEL
LIN {X 0,Y 481.755,Z 378.972,A -85,B 0,C 180,E1 -6831.612,E2 -6831.612} C_VEL
LIN {X 0,Y 481.813,Z 378.962,A -85,B 0,C 180,E1 -6834.14,E2 -6834.14} C_VEL
LIN {X 0,Y 481.926,Z 378.95,A -85,B 0,C 180,E1 -6837.493,E2 -6837.493} C_VEL
LIN {X 0,Y 481.931,Z 378.947,A -85,B 0,C 180,E1 -6840,E2 -6840} C_VEL
LIN {X 0,Y 481.92,Z 378.955,A -85,B 0,C 180,E1 -6842.508,E2 -6842.508} C_VEL
LIN {X 0,Y 481.813,Z 378.964,A -85,B 0,C 180,E1 -6845.861,E2 -6845.861} C_VEL
LIN {X 0,Y 481.755,Z 378.973,A -85,B 0,C 180,E1 -6848.389,E2 -6848.389} C_VEL
LIN {X 0,Y 481.786,Z 378.967,A -85,B 0,C 180,E1 -6851.784,E2 -6851.784} C_VEL
LIN {X 0,Y 481.733,Z 378.976,A -85,B 0,C 180,E1 -6855.225,E2 -6855.225} C_VEL
LIN {X 0,Y 481.704,Z 378.981,A -85,B 0,C 180,E1 -6858.722,E2 -6858.722} C_VEL
LIN {X 0,Y 481.646,Z 378.984,A -85,B 0,C 180,E1 -6861.395,E2 -6861.395} C_VEL
LIN {X 0,Y 481.674,Z 378.982,A -85,B 0,C 180,E1 -6864.113,E2 -6864.113} C_VEL
LIN {X 0,Y 481.744,Z 378.974,A -85,B 0,C 180,E1 -6867.141,E2 -6867.141} C_VEL
LIN {X 0,Y 481.672,Z 378.981,A -85,B 0,C 180,E1 -6869.742,E2 -6869.742} C_VEL
LIN {X 0,Y 481.666,Z 378.989,A -85,B 0,C 180,E1 -6872.675,E2 -6872.675} C_VEL
LIN {X 0,Y 481.637,Z 378.987,A -85,B 0,C 180,E1 -6875.71,E2 -6875.71} C_VEL
LIN {X 0,Y 481.709,Z 378.977,A -85,B 0,C 180,E1 -6879.355,E2 -6879.355} C_VEL
LIN {X 0,Y 481.67,Z 378.976,A -85,B 0,C 180,E1 -6882.159,E2 -6882.159} C_VEL
LIN {X 0,Y 481.656,Z 378.992,A -85,B 0,C 180,E1 -6884.458,E2 -6884.458} C_VEL
LIN {X 0,Y 481.65,Z 378.985,A -85,B 0,C 180,E1 -6887.841,E2 -6887.841} C_VEL
LIN {X 0,Y 481.678,Z 378.984,A -85,B 0,C 180,E1 -6890.652,E2 -6890.652} C_VEL
LIN {X 0,Y 481.63,Z 378.984,A -85,B 0,C 180,E1 -6893.376,E2 -6893.376} C_VEL
LIN {X 0,Y 481.708,Z 378.981,A -85,B 0,C 180,E1 -6896.331,E2 -6896.331} C_VEL
LIN {X 0,Y 481.651,Z 378.987,A -85,B 0,C 180,E1 -6899.418,E2 -6899.418} C_VEL
LIN {X 0,Y 481.702,Z 378.983,A -85,B 0,C 180,E1 -6902.169,E2 -6902.169} C_VEL
LIN {X 0,Y 481.757,Z 379.127,A -85,B 0,C 180,E1 -6905.376,E2 -6905.376} C_VEL
LIN {X 0,Y 483.516,Z 388.805,A -85,B 0,C 180,E1 -6907.346,E2 -6907.346} C_VEL
LIN {X 0,Y 483.505,Z 393.488,A -85,B 0,C 180,E1 -6908.226,E2 -6908.226} C_VEL
LIN {X 0,Y 482.717,Z 412.76,A -85,B 0,C 180,E1 -6911.759,E2 -6911.759} C_VEL
LIN {X 0,Y 482.401,Z 422.397,A -85,B 0,C 180,E1 -6913.452,E2 -6913.452} C_VEL
LIN {X 0,Y 484.943,Z 438.847,A -85,B 0,C 180,E1 -6913.818,E2 -6913.818} C_VEL
LIN {X 0,Y 484.326,Z 530.11,A -85,B 0,C 180,E1 -6915.209,E2 -6915.209} C_VEL
LIN {X 0,Y 483.962,Z 543.345,A -85,B 0,C 180,E1 -6915.574,E2 -6915.574} C_VEL
LIN {X 0,Y 483.604,Z 555.484,A -85,B 0,C 180,E1 -6916.073,E2 -6916.073} C_VEL
LIN {X 0,Y 483.235,Z 566.228,A -85,B 0,C 180,E1 -6916.662,E2 -6916.662} C_VEL
LIN {X 0,Y 482.759,Z 578.027,A -85,B 0,C 180,E1 -6917.494,E2 -6917.494} C_VEL
LIN {X 0,Y 482.344,Z 588.676,A -85,B 0,C 180,E1 -6918.443,E2 -6918.443} C_VEL
LIN {X 0,Y 481.879,Z 598.272,A -85,B 0,C 180,E1 -6919.496,E2 -6919.496} C_VEL
LIN {X 0,Y 481.586,Z 606.145,A -85,B 0,C 180,E1 -6920.551,E2 -6920.551} C_VEL
LIN {X 0,Y 481.261,Z 613.833,A -85,B 0,C 180,E1 -6921.815,E2 -6921.815} C_VEL
LIN {X 0,Y 481.048,Z 620.919,A -85,B 0,C 180,E1 -6923.288,E2 -6923.288} C_VEL
LIN {X 0,Y 480.964,Z 625.633,A -85,B 0,C 180,E1 -6924.55,E2 -6924.55} C_VEL
LIN {X 0,Y 480.829,Z 629.234,A -85,B 0,C 180,E1 -6925.809,E2 -6925.809} C_VEL
LIN {X 0,Y 480.871,Z 631.093,A -85,B 0,C 180,E1 -6926.649,E2 -6926.649} C_VEL
LIN {X 0,Y 480.789,Z 633.481,A -85,B 0,C 180,E1 -6928.325,E2 -6928.325} C_VEL
LIN {X 0,Y 480.76,Z 634.089,A -85,B 0,C 180,E1 -6929.163,E2 -6929.163} C_VEL
LIN {X 0,Y 480.743,Z 634.305,A -85,B 0,C 180,E1 -6930,E2 -6930} C_VEL
LIN {X 0,Y 480.79,Z 633.487,A -85,B 0,C 180,E1 -6931.675,E2 -6931.675} C_VEL
LIN {X 0,Y 480.871,Z 631.104,A -85,B 0,C 180,E1 -6933.352,E2 -6933.352} C_VEL
LIN {X 0,Y 480.841,Z 628.176,A -85,B 0,C 180,E1 -6934.611,E2 -6934.611} C_VEL
LIN {X 0,Y 480.967,Z 624.212,A -85,B 0,C 180,E1 -6935.871,E2 -6935.871} C_VEL
LIN {X 0,Y 481.112,Z 618.111,A -85,B 0,C 180,E1 -6937.344,E2 -6937.344} C_VEL
LIN {X 0,Y 481.369,Z 611.442,A -85,B 0,C 180,E1 -6938.607,E2 -6938.607} C_VEL
LIN {X 0,Y 481.701,Z 603.165,A -85,B 0,C 180,E1 -6939.871,E2 -6939.871} C_VEL
LIN {X 0,Y 482.048,Z 594.673,A -85,B 0,C 180,E1 -6940.926,E2 -6940.926} C_VEL
LIN {X 0,Y 482.553,Z 584.178,A -85,B 0,C 180,E1 -6941.978,E2 -6941.978} C_VEL
LIN {X 0,Y 482.92,Z 573.784,A -85,B 0,C 180,E1 -6942.822,E2 -6942.822} C_VEL
LIN {X 0,Y 483.327,Z 562.368,A -85,B 0,C 180,E1 -6943.56,E2 -6943.56} C_VEL
LIN {X 0,Y 483.775,Z 550.609,A -85,B 0,C 180,E1 -6944.137,E2 -6944.137} C_VEL
LIN {X 0,Y 484.095,Z 537.955,A -85,B 0,C 180,E1 -6944.584,E2 -6944.584} C_VEL
LIN {X 0,Y 484.336,Z 525,A -85,B 0,C 180,E1 -6944.872,E2 -6944.872} C_VEL
LIN {X 0,Y 484.81,Z 437.295,A -85,B 0,C 180,E1 -6946.18,E2 -6946.18} C_VEL
LIN {X 0,Y 482.364,Z 422.438,A -85,B 0,C 180,E1 -6946.506,E2 -6946.506} C_VEL
LIN {X 0,Y 482.928,Z 405.293,A -85,B 0,C 180,E1 -6949.555,E2 -6949.555} C_VEL
LIN {X 0,Y 483.531,Z 389.501,A -85,B 0,C 180,E1 -6952.429,E2 -6952.429} C_VEL
LIN {X 0,Y 481.75,Z 379.176,A -85,B 0,C 180,E1 -6954.453,E2 -6954.453} C_VEL
LIN {X 0,Y 481.748,Z 378.978,A -85,B 0,C 180,E1 -6957.139,E2 -6957.139} C_VEL
LIN {X 0,Y 481.68,Z 378.985,A -85,B 0,C 180,E1 -6959.741,E2 -6959.741} C_VEL
LIN {X 0,Y 481.674,Z 378.982,A -85,B 0,C 180,E1 -6962.674,E2 -6962.674} C_VEL
LIN {X 0,Y 481.643,Z 378.989,A -85,B 0,C 180,E1 -6965.708,E2 -6965.708} C_VEL
LIN {X 0,Y 481.671,Z 378.984,A -85,B 0,C 180,E1 -6968.858,E2 -6968.858} C_VEL
LIN {X 0,Y 481.661,Z 378.985,A -85,B 0,C 180,E1 -6971.914,E2 -6971.914} C_VEL
LIN {X 0,Y 481.658,Z 378.985,A -85,B 0,C 180,E1 -6974.457,E2 -6974.457} C_VEL
LIN {X 0,Y 481.687,Z 378.983,A -85,B 0,C 180,E1 -6976.845,E2 -6976.845} C_VEL
LIN {X 0,Y 481.691,Z 378.981,A -85,B 0,C 180,E1 -6980.061,E2 -6980.061} C_VEL
LIN {X 0,Y 481.627,Z 378.994,A -85,B 0,C 180,E1 -6983.253,E2 -6983.253} C_VEL
LIN {X 0,Y 481.706,Z 378.98,A -85,B 0,C 180,E1 -6986.33,E2 -6986.33} C_VEL
LIN {X 0,Y 481.647,Z 378.989,A -85,B 0,C 180,E1 -6989.417,E2 -6989.417} C_VEL
LIN {X 0,Y 481.697,Z 378.981,A -85,B 0,C 180,E1 -6992.168,E2 -6992.168} C_VEL
LIN {X 0,Y 481.714,Z 378.983,A -85,B 0,C 180,E1 -6994.97,E2 -6994.97} C_VEL
LIN {X 0,Y 481.644,Z 378.987,A -85,B 0,C 180,E1 -6997.704,E2 -6997.704} C_VEL
LIN {X 0,Y 481.703,Z 378.982,A -85,B 0,C 180,E1 -7000.393,E2 -7000.393} C_VEL
LIN {X 0,Y 481.686,Z 378.986,A -85,B 0,C 180,E1 -7003.034,E2 -7003.034} C_VEL
LIN {X 0,Y 481.683,Z 378.983,A -85,B 0,C 180,E1 -7005.638,E2 -7005.638} C_VEL
LIN {X 0,Y 481.744,Z 378.977,A -85,B 0,C 180,E1 -7008.215,E2 -7008.215} C_VEL
LIN {X 0,Y 481.757,Z 378.974,A -85,B 0,C 180,E1 -7011.612,E2 -7011.612} C_VEL
LIN {X 0,Y 481.81,Z 378.969,A -85,B 0,C 180,E1 -7014.139,E2 -7014.139} C_VEL
LIN {X 0,Y 481.922,Z 378.953,A -85,B 0,C 180,E1 -7017.492,E2 -7017.492} C_VEL
LIN {X 0,Y 481.9,Z 378.958,A -85,B 0,C 180,E1 -7020.836,E2 -7020.836} C_VEL
LIN {X 0,Y 481.922,Z 378.956,A -85,B 0,C 180,E1 -7022.507,E2 -7022.507} C_VEL
LIN {X 0,Y 481.81,Z 378.97,A -85,B 0,C 180,E1 -7025.86,E2 -7025.86} C_VEL
LIN {X 0,Y 481.756,Z 378.976,A -85,B 0,C 180,E1 -7028.388,E2 -7028.388} C_VEL
LIN {X 0,Y 481.744,Z 378.979,A -85,B 0,C 180,E1 -7031.785,E2 -7031.785} C_VEL
LIN {X 0,Y 481.736,Z 378.976,A -85,B 0,C 180,E1 -7035.224,E2 -7035.224} C_VEL
LIN {X 0,Y 481.707,Z 378.981,A -85,B 0,C 180,E1 -7038.722,E2 -7038.722} C_VEL
LIN {X 0,Y 481.641,Z 378.989,A -85,B 0,C 180,E1 -7041.395,E2 -7041.395} C_VEL
LIN {X 0,Y 481.672,Z 378.986,A -85,B 0,C 180,E1 -7044.113,E2 -7044.113} C_VEL
LIN {X 0,Y 481.747,Z 378.975,A -85,B 0,C 180,E1 -7047.141,E2 -7047.141} C_VEL
LIN {X 0,Y 481.683,Z 378.986,A -85,B 0,C 180,E1 -7049.741,E2 -7049.741} C_VEL
LIN {X 0,Y 481.669,Z 378.984,A -85,B 0,C 180,E1 -7052.674,E2 -7052.674} C_VEL
LIN {X 0,Y 481.639,Z 378.991,A -85,B 0,C 180,E1 -7055.709,E2 -7055.709} C_VEL
LIN {X 0,Y 481.668,Z 378.985,A -85,B 0,C 180,E1 -7058.859,E2 -7058.859} C_VEL
LIN {X 0,Y 481.659,Z 378.987,A -85,B 0,C 180,E1 -7061.915,E2 -7061.915} C_VEL
LIN {X 0,Y 481.657,Z 378.985,A -85,B 0,C 180,E1 -7064.458,E2 -7064.458} C_VEL
LIN {X 0,Y 481.646,Z 378.988,A -85,B 0,C 180,E1 -7067.84,E2 -7067.84} C_VEL
LIN {X 0,Y 481.713,Z 378.978,A -85,B 0,C 180,E1 -7070.647,E2 -7070.647} C_VEL
LIN {X 0,Y 481.642,Z 378.987,A -85,B 0,C 180,E1 -7074.292,E2 -7074.292} C_VEL
LIN {X 0,Y 481.672,Z 378.988,A -85,B 0,C 180,E1 -7077.326,E2 -7077.326} C_VEL
LIN {X 0,Y 481.679,Z 378.982,A -85,B 0,C 180,E1 -7080.259,E2 -7080.259} C_VEL
LIN {X 0,Y 481.746,Z 378.98,A -85,B 0,C 180,E1 -7083.112,E2 -7083.112} C_VEL
LIN {X 0,Y 481.675,Z 378.983,A -85,B 0,C 180,E1 -7085.887,E2 -7085.887} C_VEL
LIN {X 0,Y 481.636,Z 378.987,A -85,B 0,C 180,E1 -7087.991,E2 -7087.991} C_VEL
LIN {X 0,Y 480.969,Z 379.074,A -85,B 0,C 180,E1 -7088.689,E2 -7088.689} C_VEL
LIN {X 0,Y 478.143,Z 379.424,A -85,B 0,C 180,E1 -7089.823,E2 -7089.823} C_VEL
LIN {X 0,Y 475.758,Z 379.722,A -85,B 0,C 180,E1 -7090.737,E2 -7090.737} C_VEL
LIN {X 0,Y 474.738,Z 379.849,A -85,B 0,C 180,E1 -7091.443,E2 -7091.443} C_VEL
LIN {X 0,Y 474.656,Z 379.857,A -85,B 0,C 180,E1 -7091.682,E2 -7091.682} C_VEL
LIN {X 0,Y 474.702,Z 379.852,A -85,B 0,C 180,E1 -7094.545,E2 -7094.545} C_VEL
LIN {X 0,Y 474.706,Z 379.853,A -85,B 0,C 180,E1 -7098.038,E2 -7098.038} C_VEL
LIN {X 0,Y 474.731,Z 380.066,A -85,B 0,C 180,E1 -7100.252,E2 -7100.252} C_VEL
LIN {X 0,Y 476.094,Z 387.603,A -85,B 0,C 180,E1 -7101.874,E2 -7101.874} C_VEL
LIN {X 0,Y 475.741,Z 397.432,A -85,B 0,C 180,E1 -7103.852,E2 -7103.852} C_VEL
LIN {X 0,Y 475.391,Z 409.857,A -85,B 0,C 180,E1 -7106.291,E2 -7106.291} C_VEL
LIN {X 0,Y 476.194,Z 414.496,A -85,B 0,C 180,E1 -7106.43,E2 -7106.43} C_VEL
LIN {X 0,Y 478.096,Z 425.061,A -85,B 0,C 180,E1 -7106.655,E2 -7106.655} C_VEL
LIN {X 0,Y 477.392,Z 517.573,A -85,B 0,C 180,E1 -7108.075,E2 -7108.075} C_VEL
LIN {X 0,Y 477.083,Z 531.25,A -85,B 0,C 180,E1 -7108.47,E2 -7108.47} C_VEL
LIN {X 0,Y 476.751,Z 543.53,A -85,B 0,C 180,E1 -7108.997,E2 -7108.997} C_VEL
LIN {X 0,Y 476.265,Z 555.35,A -85,B 0,C 180,E1 -7109.683,E2 -7109.683} C_VEL
LIN {X 0,Y 475.743,Z 566.693,A -85,B 0,C 180,E1 -7110.529,E2 -7110.529} C_VEL
LIN {X 0,Y 475.3,Z 576.922,A -85,B 0,C 180,E1 -7111.483,E2 -7111.483} C_VEL
LIN {X 0,Y 474.838,Z 586.144,A -85,B 0,C 180,E1 -7112.545,E2 -7112.545} C_VEL
LIN {X 0,Y 474.451,Z 595.09,A -85,B 0,C 180,E1 -7113.822,E2 -7113.822} C_VEL
LIN {X 0,Y 474.087,Z 602.331,A -85,B 0,C 180,E1 -7115.103,E2 -7115.103} C_VEL
LIN {X 0,Y 473.997,Z 608.86,A -85,B 0,C 180,E1 -7116.579,E2 -7116.579} C_VEL
LIN {X 0,Y 473.824,Z 613.95,A -85,B 0,C 180,E1 -7118.1,E2 -7118.1} C_VEL
LIN {X 0,Y 473.68,Z 617.102,A -85,B 0,C 180,E1 -7119.393,E2 -7119.393} C_VEL
LIN {X 0,Y 473.673,Z 618.668,A -85,B 0,C 180,E1 -7120.256,E2 -7120.256} C_VEL
LIN {X 0,Y 473.706,Z 620.321,A -85,B 0,C 180,E1 -7121.709,E2 -7121.709} C_VEL
LIN {X 0,Y 473.649,Z 620.786,A -85,B 0,C 180,E1 -7122.86,E2 -7122.86} C_VEL
LIN {X 0,Y 473.6,Z 620.688,A -85,B 0,C 180,E1 -7123.735,E2 -7123.735} C_VEL
LIN {X 0,Y 473.661,Z 619.378,A -85,B 0,C 180,E1 -7125.324,E2 -7125.324} C_VEL
LIN {X 0,Y 473.653,Z 617.77,A -85,B 0,C 180,E1 -7126.374,E2 -7126.374} C_VEL
LIN {X 0,Y 473.789,Z 614.793,A -85,B 0,C 180,E1 -7127.703,E2 -7127.703} C_VEL
LIN {X 0,Y 473.908,Z 610.682,A -85,B 0,C 180,E1 -7129.041,E2 -7129.041} C_VEL
LIN {X 0,Y 474.129,Z 604.22,A -85,B 0,C 180,E1 -7130.612,E2 -7130.612} C_VEL
LIN {X 0,Y 474.434,Z 597.078,A -85,B 0,C 180,E1 -7131.964,E2 -7131.964} C_VEL
LIN {X 0,Y 474.781,Z 589.84,A -85,B 0,C 180,E1 -7133.074,E2 -7133.074} C_VEL
LIN {X 0,Y 475.195,Z 580.623,A -85,B 0,C 180,E1 -7134.23,E2 -7134.23} C_VEL
LIN {X 0,Y 475.63,Z 570.523,A -85,B 0,C 180,E1 -7135.255,E2 -7135.255} C_VEL
LIN {X 0,Y 476.167,Z 559.056,A -85,B 0,C 180,E1 -7136.187,E2 -7136.187} C_VEL
LIN {X 0,Y 476.597,Z 547.74,A -85,B 0,C 180,E1 -7136.905,E2 -7136.905} C_VEL
LIN {X 0,Y 477.048,Z 535.5,A -85,B 0,C 180,E1 -7137.492,E2 -7137.492} C_VEL
LIN {X 0,Y 477.367,Z 522.346,A -85,B 0,C 180,E1 -7137.939,E2 -7137.939} C_VEL
LIN {X 0,Y 477.569,Z 508.604,A -85,B 0,C 180,E1 -7138.213,E2 -7138.213} C_VEL
LIN {X 0,Y 478.151,Z 424.663,A -85,B 0,C 180,E1 -7139.493,E2 -7139.493} C_VEL
LIN {X 0,Y 475.5,Z 410.435,A -85,B 0,C 180,E1 -7139.831,E2 -7139.831} C_VEL
LIN {X 0,Y 475.454,Z 409.534,A -85,B 0,C 180,E1 -7139.919,E2 -7139.919} C_VEL
LIN {X 0,Y 476.209,Z 392.475,A -85,B 0,C 180,E1 -7143.348,E2 -7143.348} C_VEL
LIN {X 0,Y 476.199,Z 388.074,A -85,B 0,C 180,E1 -7144.261,E2 -7144.261} C_VEL
LIN {X 0,Y 474.642,Z 379.931,A -85,B 0,C 180,E1 -7146.105,E2 -7146.105} C_VEL
LIN {X 0,Y 474.651,Z 379.862,A -85,B 0,C 180,E1 -7149.651,E2 -7149.651} C_VEL
LIN {X 0,Y 474.648,Z 379.861,A -85,B 0,C 180,E1 -7152.929,E2 -7152.929} C_VEL
LIN {X 0,Y 474.613,Z 379.863,A -85,B 0,C 180,E1 -7155.895,E2 -7155.895} C_VEL
LIN {X 0,Y 474.641,Z 379.862,A -85,B 0,C 180,E1 -7159.037,E2 -7159.037} C_VEL
LIN {X 0,Y 474.614,Z 379.861,A -85,B 0,C 180,E1 -7161.702,E2 -7161.702} C_VEL
LIN {X 0,Y 474.624,Z 379.862,A -85,B 0,C 180,E1 -7164.726,E2 -7164.726} C_VEL
LIN {X 0,Y 474.63,Z 379.86,A -85,B 0,C 180,E1 -7167.787,E2 -7167.787} C_VEL
LIN {X 0,Y 474.624,Z 379.856,A -85,B 0,C 180,E1 -7170.882,E2 -7170.882} C_VEL
LIN {X 0,Y 474.658,Z 379.857,A -85,B 0,C 180,E1 -7173.628,E2 -7173.628} C_VEL
LIN {X 0,Y 474.628,Z 379.864,A -85,B 0,C 180,E1 -7176.641,E2 -7176.641} C_VEL
LIN {X 0,Y 474.667,Z 379.86,A -85,B 0,C 180,E1 -7179.185,E2 -7179.185} C_VEL
LIN {X 0,Y 474.648,Z 379.854,A -85,B 0,C 180,E1 -7181.884,E2 -7181.884} C_VEL
LIN {X 0,Y 474.69,Z 379.855,A -85,B 0,C 180,E1 -7184.544,E2 -7184.544} C_VEL
LIN {X 0,Y 474.729,Z 379.847,A -85,B 0,C 180,E1 -7188.038,E2 -7188.038} C_VEL
LIN {X 0,Y 474.72,Z 379.849,A -85,B 0,C 180,E1 -7191.486,E2 -7191.486} C_VEL
LIN {X 0,Y 474.775,Z 379.838,A -85,B 0,C 180,E1 -7194.052,E2 -7194.052} C_VEL
LIN {X 0,Y 474.892,Z 379.826,A -85,B 0,C 180,E1 -7197.455,E2 -7197.455} C_VEL
LIN {X 0,Y 474.869,Z 379.836,A -85,B 0,C 180,E1 -7200.848,E2 -7200.848} C_VEL
LIN {X 0,Y 474.887,Z 379.832,A -85,B 0,C 180,E1 -7202.545,E2 -7202.545} C_VEL
LIN {X 0,Y 474.775,Z 379.841,A -85,B 0,C 180,E1 -7205.948,E2 -7205.948} C_VEL
LIN {X 0,Y 474.72,Z 379.851,A -85,B 0,C 180,E1 -7208.514,E2 -7208.514} C_VEL
LIN {X 0,Y 474.73,Z 379.847,A -85,B 0,C 180,E1 -7211.962,E2 -7211.962} C_VEL
LIN {X 0,Y 474.671,Z 379.854,A -85,B 0,C 180,E1 -7215.768,E2 -7215.768} C_VEL
LIN {X 0,Y 474.657,Z 379.859,A -85,B 0,C 180,E1 -7219.011,E2 -7219.011} C_VEL
LIN {X 0,Y 474.589,Z 379.862,A -85,B 0,C 180,E1 -7221.729,E2 -7221.729} C_VEL
LIN {X 0,Y 474.654,Z 379.86,A -85,B 0,C 180,E1 -7224.493,E2 -7224.493} C_VEL
LIN {X 0,Y 474.691,Z 379.851,A -85,B 0,C 180,E1 -7227.339,E2 -7227.339} C_VEL
LIN {X 0,Y 474.598,Z 379.867,A -85,B 0,C 180,E1 -7230.811,E2 -7230.811} C_VEL
LIN {X 0,Y 474.632,Z 379.859,A -85,B 0,C 180,E1 -7233.985,E2 -7233.985} C_VEL
LIN {X 0,Y 474.57,Z 379.869,A -85,B 0,C 180,E1 -7236.901,E2 -7236.901} C_VEL
LIN {X 0,Y 474.645,Z 379.857,A -85,B 0,C 180,E1 -7239.652,E2 -7239.652} C_VEL
LIN {X 0,Y 474.648,Z 379.861,A -85,B 0,C 180,E1 -7242.931,E2 -7242.931} C_VEL
LIN {X 0,Y 474.611,Z 379.86,A -85,B 0,C 180,E1 -7245.897,E2 -7245.897} C_VEL
LIN {X 0,Y 474.629,Z 379.86,A -85,B 0,C 180,E1 -7249.041,E2 -7249.041} C_VEL
LIN {X 0,Y 474.608,Z 379.863,A -85,B 0,C 180,E1 -7251.705,E2 -7251.705} C_VEL
LIN {X 0,Y 474.629,Z 379.865,A -85,B 0,C 180,E1 -7254.727,E2 -7254.727} C_VEL
LIN {X 0,Y 474.637,Z 379.861,A -85,B 0,C 180,E1 -7257.789,E2 -7257.789} C_VEL
LIN {X 0,Y 474.624,Z 379.865,A -85,B 0,C 180,E1 -7260.885,E2 -7260.885} C_VEL
LIN {X 0,Y 474.667,Z 379.86,A -85,B 0,C 180,E1 -7263.63,E2 -7263.63} C_VEL
LIN {X 0,Y 474.719,Z 380.068,A -85,B 0,C 180,E1 -7265.161,E2 -7265.161} C_VEL
LIN {X 0,Y 476.581,Z 390.05,A -85,B 0,C 180,E1 -7267.226,E2 -7267.226} C_VEL
LIN {X 0,Y 476.618,Z 393.864,A -85,B 0,C 180,E1 -7267.959,E2 -7267.959} C_VEL
LIN {X 0,Y 475.765,Z 412.774,A -85,B 0,C 180,E1 -7271.483,E2 -7271.483} C_VEL
LIN {X 0,Y 475.407,Z 422.325,A -85,B 0,C 180,E1 -7273.188,E2 -7273.188} C_VEL
LIN {X 0,Y 478.161,Z 439.382,A -85,B 0,C 180,E1 -7273.582,E2 -7273.582} C_VEL
LIN {X 0,Y 477.484,Z 530.446,A -85,B 0,C 180,E1 -7274.992,E2 -7274.992} C_VEL
LIN {X 0,Y 477.083,Z 544.285,A -85,B 0,C 180,E1 -7275.389,E2 -7275.389} C_VEL
LIN {X 0,Y 476.692,Z 556.69,A -85,B 0,C 180,E1 -7275.921,E2 -7275.921} C_VEL
LIN {X 0,Y 476.262,Z 567.77,A -85,B 0,C 180,E1 -7276.561,E2 -7276.561} C_VEL
LIN {X 0,Y 475.767,Z 579.361,A -85,B 0,C 180,E1 -7277.419,E2 -7277.419} C_VEL
LIN {X 0,Y 475.329,Z 589.716,A -85,B 0,C 180,E1 -7278.379,E2 -7278.379} C_VEL
LIN {X 0,Y 474.883,Z 598.224,A -85,B 0,C 180,E1 -7279.34,E2 -7279.34} C_VEL
LIN {X 0,Y 474.543,Z 606.08,A -85,B 0,C 180,E1 -7280.409,E2 -7280.409} C_VEL
LIN {X 0,Y 474.221,Z 613.755,A -85,B 0,C 180,E1 -7281.692,E2 -7281.692} C_VEL
LIN {X 0,Y 473.977,Z 620.833,A -85,B 0,C 180,E1 -7283.188,E2 -7283.188} C_VEL
LIN {X 0,Y 473.879,Z 625.542,A -85,B 0,C 180,E1 -7284.468,E2 -7284.468} C_VEL
LIN {X 0,Y 473.736,Z 629.139,A -85,B 0,C 180,E1 -7285.746,E2 -7285.746} C_VEL
LIN {X 0,Y 473.765,Z 630.996,A -85,B 0,C 180,E1 -7286.599,E2 -7286.599} C_VEL
LIN {X 0,Y 473.723,Z 632.388,A -85,B 0,C 180,E1 -7287.449,E2 -7287.449} C_VEL
LIN {X 0,Y 473.688,Z 633.99,A -85,B 0,C 180,E1 -7289.15,E2 -7289.15} C_VEL
LIN {X 0,Y 473.669,Z 634.205,A -85,B 0,C 180,E1 -7290,E2 -7290} C_VEL
LIN {X 0,Y 473.688,Z 633.99,A -85,B 0,C 180,E1 -7290.85,E2 -7290.85} C_VEL
LIN {X 0,Y 473.723,Z 632.392,A -85,B 0,C 180,E1 -7292.551,E2 -7292.551} C_VEL
LIN {X 0,Y 473.765,Z 630.999,A -85,B 0,C 180,E1 -7293.402,E2 -7293.402} C_VEL
LIN {X 0,Y 473.765,Z 628.069,A -85,B 0,C 180,E1 -7294.68,E2 -7294.68} C_VEL
LIN {X 0,Y 473.87,Z 624.1,A -85,B 0,C 180,E1 -7295.959,E2 -7295.959} C_VEL
LIN {X 0,Y 474.033,Z 617.989,A -85,B 0,C 180,E1 -7297.454,E2 -7297.454} C_VEL
LIN {X 0,Y 474.336,Z 611.312,A -85,B 0,C 180,E1 -7298.735,E2 -7298.735} C_VEL
LIN {X 0,Y 474.655,Z 603.022,A -85,B 0,C 180,E1 -7300.019,E2 -7300.019} C_VEL
LIN {X 0,Y 475.072,Z 594.512,A -85,B 0,C 180,E1 -7301.088,E2 -7301.088} C_VEL
LIN {X 0,Y 475.582,Z 584.006,A -85,B 0,C 180,E1 -7302.155,E2 -7302.155} C_VEL
LIN {X 0,Y 476.035,Z 572.639,A -85,B 0,C 180,E1 -7303.082,E2 -7303.082} C_VEL
LIN {X 0,Y 476.408,Z 562.116,A -85,B 0,C 180,E1 -7303.761,E2 -7303.761} C_VEL
LIN {X 0,Y 476.889,Z 550.281,A -85,B 0,C 180,E1 -7304.345,E2 -7304.345} C_VEL
LIN {X 0,Y 477.222,Z 537.522,A -85,B 0,C 180,E1 -7304.798,E2 -7304.798} C_VEL
LIN {X 0,Y 477.462,Z 524.341,A -85,B 0,C 180,E1 -7305.091,E2 -7305.091} C_VEL
LIN {X 0,Y 478.038,Z 438.42,A -85,B 0,C 180,E1 -7306.388,E2 -7306.388} C_VEL
LIN {X 0,Y 475.384,Z 422.672,A -85,B 0,C 180,E1 -7306.728,E2 -7306.728} C_VEL
LIN {X 0,Y 475.363,Z 421.509,A -85,B 0,C 180,E1 -7306.867,E2 -7306.867} C_VEL
LIN {X 0,Y 475.967,Z 405.107,A -85,B 0,C 180,E1 -7309.853,E2 -7309.853} C_VEL
LIN {X 0,Y 476.569,Z 390.523,A -85,B 0,C 180,E1 -7312.546,E2 -7312.546} C_VEL
LIN {X 0,Y 474.682,Z 379.975,A -85,B 0,C 180,E1 -7314.666,E2 -7314.666} C_VEL
LIN {X 0,Y 474.7,Z 379.858,A -85,B 0,C 180,E1 -7317.338,E2 -7317.338} C_VEL
LIN {X 0,Y 474.606,Z 379.864,A -85,B 0,C 180,E1 -7320.81,E2 -7320.81} C_VEL
LIN {X 0,Y 474.638,Z 379.86,A -85,B 0,C 180,E1 -7323.983,E2 -7323.983} C_VEL
LIN {X 0,Y 474.576,Z 379.868,A -85,B 0,C 180,E1 -7326.9,E2 -7326.9} C_VEL
LIN {X 0,Y 474.627,Z 379.864,A -85,B 0,C 180,E1 -7329.647,E2 -7329.647} C_VEL
LIN {X 0,Y 474.634,Z 379.862,A -85,B 0,C 180,E1 -7332.931,E2 -7332.931} C_VEL
LIN {X 0,Y 474.616,Z 379.863,A -85,B 0,C 180,E1 -7335.896,E2 -7335.896} C_VEL
LIN {X 0,Y 474.645,Z 379.862,A -85,B 0,C 180,E1 -7339.037,E2 -7339.037} C_VEL
LIN {X 0,Y 474.616,Z 379.863,A -85,B 0,C 180,E1 -7341.702,E2 -7341.702} C_VEL
LIN {X 0,Y 474.626,Z 379.863,A -85,B 0,C 180,E1 -7344.726,E2 -7344.726} C_VEL
LIN {X 0,Y 474.633,Z 379.861,A -85,B 0,C 180,E1 -7347.787,E2 -7347.787} C_VEL
LIN {X 0,Y 474.62,Z 379.865,A -85,B 0,C 180,E1 -7350.884,E2 -7350.884} C_VEL
LIN {X 0,Y 474.662,Z 379.858,A -85,B 0,C 180,E1 -7353.628,E2 -7353.628} C_VEL
LIN {X 0,Y 474.63,Z 379.863,A -85,B 0,C 180,E1 -7356.641,E2 -7356.641} C_VEL
LIN {X 0,Y 474.651,Z 379.86,A -85,B 0,C 180,E1 -7360.089,E2 -7360.089} C_VEL
LIN {X 0,Y 474.646,Z 379.862,A -85,B 0,C 180,E1 -7362.774,E2 -7362.774} C_VEL
